// TIA Portal V20 export
FUNCTION_BLOCK "CallEquipment"   // FB43, LAD
TITLE = CallEquipment
// Template of an equipment module. This block contains the logic and futher calls (e.g. sequences, control modules, diagnostics etc.) of the equipment module.
// It can be used out of the box but also adapted to your own needs.
// stored: IsIECCheckEnabled true, MemoryReserve 100, Namespace Unit1.Em4, SetENOAutomatically true
   VAR_INPUT
      ZoneOperationEnable { ExternalWritable := 'False'} : "LWONIK_typeSafetyZoneManualOperation";
      unitEnableControlInterfaces { ExternalWritable := 'False'} : "LAF_typeEnableControlInterfaces";
      commandExcute { ExternalWritable := 'False'} : Bool;
   END_VAR
   VAR_IN_OUT
      unitStatus : "LAF_typeUnitStatus";   // Current unit status o be used in this EM
      emFeedback : "LUC_typeEmFeedback";   // Feedback of the EM to the Unit
      unitAlarmDB : "LAF_typeAlarms";   // Summarized EM Alarms for the Unit
   END_VAR
   VAR
      instSequence { ExternalWritable := 'False'} : "Unit1.Em4.Sequence_1_Cutter";
      instCutterInitializedJob1 { ExternalWritable := 'False'} : "LAF_SelectJob";
      instCutterCycleJob2 { S7_SetPoint := 'True'} : "LAF_SelectJob";
      instCmCompensatorAxisZ { ExternalWritable := 'False'} : "LBC_AxisControl_TecPlcCn";
      instCmFeedingRollAxisB { ExternalWritable := 'False'} : "LBC_AxisControl_TecPlcCn";
      instCmElectrodeCutterAxisZ { ExternalWritable := 'False'} : "LBC_AxisControl_TecPlcCn";
      instCmPositionMovingAxisX { ExternalWritable := 'False'} : "LBC_Axis64Pos_TecPlcCn";
      instCmFeederCylinderUpDown { ExternalWritable := 'False'} : "LBC_TwoWayActuatorCn";
      instCmCompensatorSafetyPinIdlePosition { ExternalWritable := 'False'} : "LBC_DigitalSignalCn";
      instCmTabDetectSensor { ExternalWritable := 'False'} : "LBC_DigitalSignalCn";
      instCmTapeDetectSensor { ExternalWritable := 'False'} : "LBC_DigitalSignalCn";
      instCutterEpcAnalogInput { ExternalWritable := 'False'} : "LBC_AnalogInputCn";
      instCompensatorAxisControlInterlockSummary { ExternalWritable := 'False'} : "LER_AxisControl_InterlockSummary";
      instFeedingRollAxisControlInterlockSummary { ExternalWritable := 'False'} : "LER_AxisControl_InterlockSummary";
      instCutterAxisControlInterlockSummary { ExternalWritable := 'False'} : "LER_AxisControl_InterlockSummary";
      instPostionMovingAxisControlInterlockSummary { ExternalWritable := 'False'} : "LER_Axis64Pos_InterlockSummary";
      instServoTorqueCal_DR3 { ExternalWritable := 'False'} : "LER_ServoTorqueCal";
      instServoTorqueCal_DR4 { ExternalWritable := 'False'} : "LER_ServoTorqueCal";
      instServoTorqueCal_DR5 { ExternalWritable := 'False'} : "LER_ServoTorqueCal";
      instServoTorqueCal_DR6 { ExternalWritable := 'False'} : "LER_ServoTorqueCal";
      instLDrv701ControlCompensatorAxisZ { ExternalWritable := 'False'} : "LDrvSafe_SinaTlg701Control";   // Drive Telegram Function Library
      instLDrv701StatusCompensatorAxisZ { ExternalWritable := 'False'} : "LDrvSafe_SinaTlg701Status";   // Drive Telegram Function Library
      instLDrv701ControlFeedingRollAxisB { ExternalWritable := 'False'} : "LDrvSafe_SinaTlg701Control";   // Drive Telegram Function Library
      instLDrv701StatusFeedingRollAxisB { ExternalWritable := 'False'} : "LDrvSafe_SinaTlg701Status";   // Drive Telegram Function Library
      instLDrv701ControlElectrodeCutterAxisZ { ExternalWritable := 'False'} : "LDrvSafe_SinaTlg701Control";   // Drive Telegram Function Library
      instLDrv701StatusElectrodeCutterAxisZ { ExternalWritable := 'False'} : "LDrvSafe_SinaTlg701Status";   // Drive Telegram Function Library
      instLDrv701ControlPositionMovingAxisX { ExternalWritable := 'False'} : "LDrvSafe_SinaTlg701Control";   // Drive Telegram Function Library
      instLDrv701StatusPositionMovingAxisX { ExternalWritable := 'False'} : "LDrvSafe_SinaTlg701Status";   // Drive Telegram Function Library
      statUnitStatus { ExternalWritable := 'False'} : "LAF_typeUnitStatus";   // Unit Status used in this EM
      statAllBrakeTest { ExternalWritable := 'False'} : "LER_typeBrakeTestUnitCommands";
      instManageAlarms { ExternalWritable := 'False'} : "LAF_ManageAlarms";
      instEventsPFE { S7_SetPoint := 'True'} : "Unit1.Em4.EventsPFE";
      statPulse { ExternalWritable := 'False'} : Array[0..99] of Bool;
      statTonTimer { ExternalWritable := 'False'} : Array[0..99] of TON_TIME;
      statTofTimer { ExternalWritable := 'False'} : Array[0..99] of TOF_TIME;
      statEnableManualCmds { ExternalWritable := 'False'} : Bool;
      EndOfCycle_Complete { ExternalWritable := 'False'} : Bool;
   END_VAR
   VAR_TEMP
      tempScInProduction : Bool;   // Mode Production and StateComplete
      tempScNoProduction : Bool;   // Mode Manual and StateComplete
   END_VAR
   VAR CONSTANT
      TO_DO_INSERT_PRECONDITIONS_HERE : Bool := TRUE;   // Template : Add em specific conditions here
      NO_JOB : DInt;   // No job
      TRUE : Bool := TRUE;
      FALSE : Bool := FALSE;
      "acc/dccTime" : LReal := 3.0;
      JerkTime : LReal := 0.0;
      INIT_POSITION_NUMBER : SInt := -1;
      MIN_POSITION_NUMBER : SInt;
   END_VAR
   VAR_TEMP   // added for the SCL form of the ladder/FBD networks
      _w1 : Bool;
      _w2 : Bool;
      _w3 : Bool;
      _w4 : Bool;
      _w5 : Bool;
      _w6 : Bool;
      _w7 : Bool;
      _w8 : Bool;
      _w9 : Bool;
      _w10 : Bool;
      _w11 : Bool;
      _w12 : Bool;
      _w13 : Bool;
      _w14 : Bool;
      _w15 : Bool;
      _w16 : Bool;
   END_VAR
BEGIN

REGION Network 1: BLOCK INFO HEADER
   // (company) / (C) Copyright (year)
   // ---------------------------------------------------------------------------------
   // Title:                             (Title of this block)
   // Comment/Function: (that is implemented in the block)
   // Library/Family:           (that the source is dedicated to)
   // Author:                        (department / person in charge / contact)
   // Target System:          (test system with FW version)
   // Engineering:              TIA Portal (SW version)
   // Restrictions:               (OB types, etc.)
   // Requirements:           (hardware, technological package, etc.)
   // ---------------------------------------------------------------------------------
   // Change log table:
   // Version          | Date             | Signature      | Expert in charge  | Changes applied ------------------------|----------------------|-------------------------|--------------------------------|-----------------------
   // 001.000.000 | yyyy-mm-dd | 0x00000000 | (name of expert) | First released version
END_REGION

REGION Network 2: DESCRIPTION
   // This is a template block provided by the Automation Framework. It can be used to create an own project.
   // The Block Info Header is prepared to put in your own data.
   // Description of the block could be added here and the docu created by Code2Docu.
END_REGION

REGION Network 3: ******************** Unit Input ********************
END_REGION

REGION Network 4: Em Nodes Brake Test
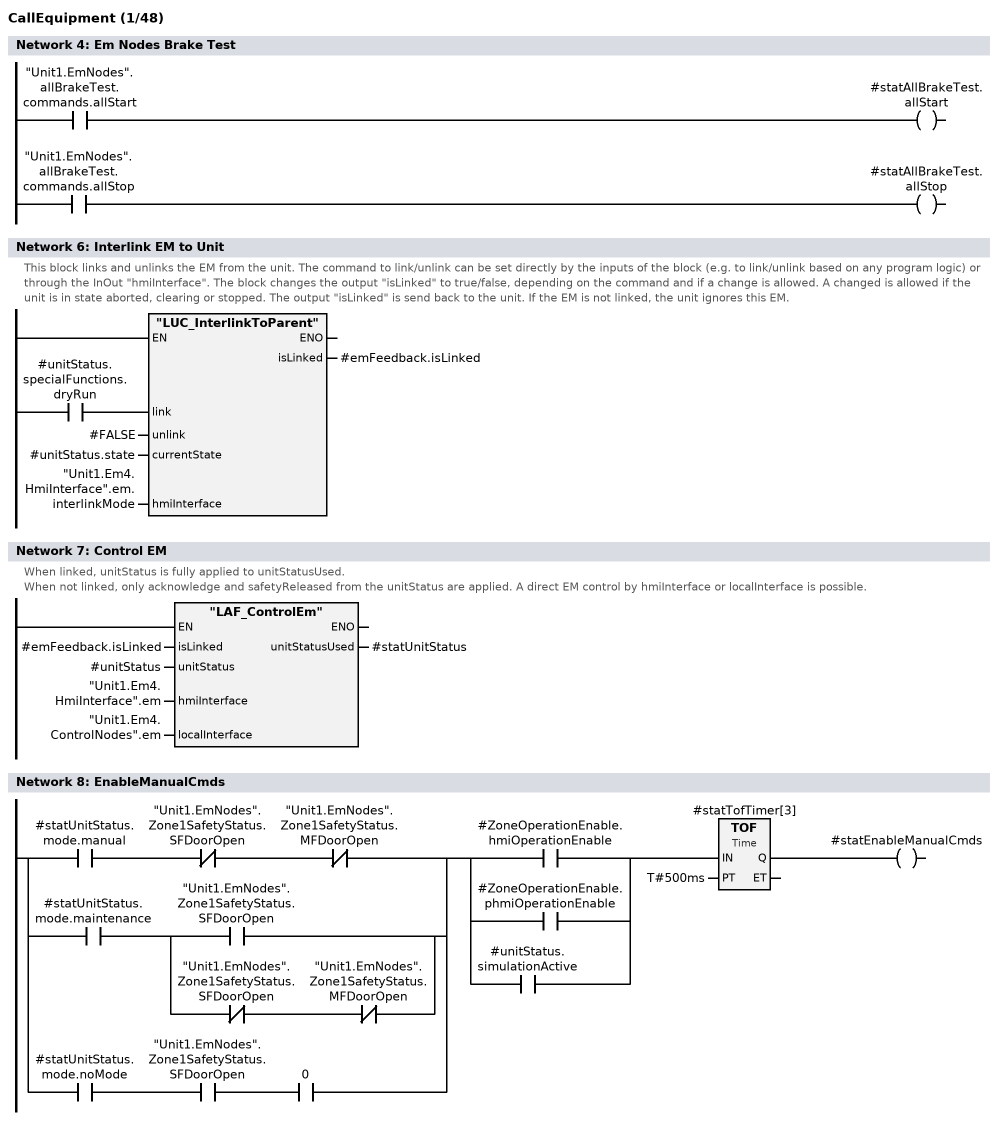
   RUNG wire#powerrail
      Contact( "Unit1.EmNodes".allBrakeTest.commands.allStart )
      Coil( #statAllBrakeTest.allStart )
   END_RUNG
   RUNG wire#powerrail
      Contact( "Unit1.EmNodes".allBrakeTest.commands.allStop )
      Coil( #statAllBrakeTest.allStop )
   END_RUNG
   // the same network as SCL:
   #statAllBrakeTest.allStart := "Unit1.EmNodes".allBrakeTest.commands.allStart;
   #statAllBrakeTest.allStop := "Unit1.EmNodes".allBrakeTest.commands.allStop;
END_REGION

REGION Network 5: ******************** Equipment Control ********************
END_REGION

REGION Network 6: Interlink EM to Unit
   // This block links and unlinks the EM from the unit. The command to link/unlink can be set directly by the inputs of the block (e.g. to link/unlink based on any program logic) or through the InOut "hmiInterface". The block changes the output "isLinked" to true/false, depending on the command and if a change is allowed. A changed is allowed if the unit is in state aborted, clearing or stopped. The output "isLinked" is send back to the unit. If the EM is not linked, the unit ignores this EM.
   RUNG wire#powerrail
      "LUC_InterlinkToParent"(link := wire#w1, unlink := #FALSE, currentState := #unitStatus.state, hmiInterface := "Unit1.Em4.HmiInterface".em.interlinkMode, isLinked => #emFeedback.isLinked)
   END_RUNG
   RUNG wire#powerrail
      Contact( #unitStatus.specialFunctions.dryRun )
   END_RUNG wire#w1
   // the same network as SCL:
   "LUC_InterlinkToParent"(link := #unitStatus.specialFunctions.dryRun,
                           unlink := #FALSE,
                           currentState := #unitStatus.state,
                           hmiInterface := "Unit1.Em4.HmiInterface".em.interlinkMode,
                           isLinked => #emFeedback.isLinked);
END_REGION

REGION Network 7: Control EM
   // When linked, unitStatus is fully applied to unitStatusUsed.
   // When not linked, only acknowledge and safetyReleased from the unitStatus are applied. A direct EM control by hmiInterface or localInterface is possible.
   RUNG wire#powerrail
      "LAF_ControlEm"(isLinked := #emFeedback.isLinked, unitStatus := #unitStatus, hmiInterface := "Unit1.Em4.HmiInterface".em, localInterface := "Unit1.Em4.ControlNodes".em, unitStatusUsed => #statUnitStatus)
   END_RUNG
   // the same network as SCL:
   "LAF_ControlEm"(isLinked := #emFeedback.isLinked,
                   unitStatus := #unitStatus,
                   hmiInterface := "Unit1.Em4.HmiInterface".em,
                   localInterface := "Unit1.Em4.ControlNodes".em,
                   unitStatusUsed => #statUnitStatus);
END_REGION

REGION Network 8: EnableManualCmds
   RUNG wire#powerrail
      Contact( #statUnitStatus.mode.manual )
      I_Contact( "Unit1.EmNodes".Zone1SafetyStatus.SFDoorOpen )
      I_Contact( "Unit1.EmNodes".Zone1SafetyStatus.MFDoorOpen )
      wire#w1
      Contact( #ZoneOperationEnable.hmiOperationEnable )
      wire#w3
      { S7_Templates := "time_type := Time" } #statTofTimer[3].TOF(pt := T#500ms, et =>)
      Coil( #statEnableManualCmds )
   END_RUNG
   RUNG wire#powerrail
      Contact( #statUnitStatus.mode.maintenance )
      wire#w2
      Contact( "Unit1.EmNodes".Zone1SafetyStatus.SFDoorOpen )
   END_RUNG wire#w1
   RUNG wire#w2
      I_Contact( "Unit1.EmNodes".Zone1SafetyStatus.SFDoorOpen )
      I_Contact( "Unit1.EmNodes".Zone1SafetyStatus.MFDoorOpen )
   END_RUNG wire#w1
   RUNG wire#powerrail
      Contact( #statUnitStatus.mode.noMode )
      Contact( "Unit1.EmNodes".Zone1SafetyStatus.SFDoorOpen )
      Contact( 0 )
   END_RUNG wire#w1
   RUNG wire#w1
      Contact( #ZoneOperationEnable.phmiOperationEnable )
   END_RUNG wire#w3
   RUNG wire#w1
      Contact( #unitStatus.simulationActive )
   END_RUNG wire#w3
   // the same network as SCL:
   #statTofTimer[3].TOF(IN := ((#statUnitStatus.mode.manual AND NOT "Unit1.EmNodes".Zone1SafetyStatus.SFDoorOpen AND NOT "Unit1.EmNodes".Zone1SafetyStatus.MFDoorOpen) OR (#statUnitStatus.mode.maintenance AND ("Unit1.EmNodes".Zone1SafetyStatus.SFDoorOpen OR (NOT "Unit1.EmNodes".Zone1SafetyStatus.SFDoorOpen AND NOT "Unit1.EmNodes".Zone1SafetyStatus.MFDoorOpen))) OR (#statUnitStatus.mode.noMode AND "Unit1.EmNodes".Zone1SafetyStatus.SFDoorOpen AND 0)) AND (#ZoneOperationEnable.hmiOperationEnable OR #ZoneOperationEnable.phmiOperationEnable OR #unitStatus.simulationActive),
                        PT := T#500ms);
   #statEnableManualCmds := #statTofTimer[3].Q;
END_REGION

REGION Network 9: Alarms Disabled
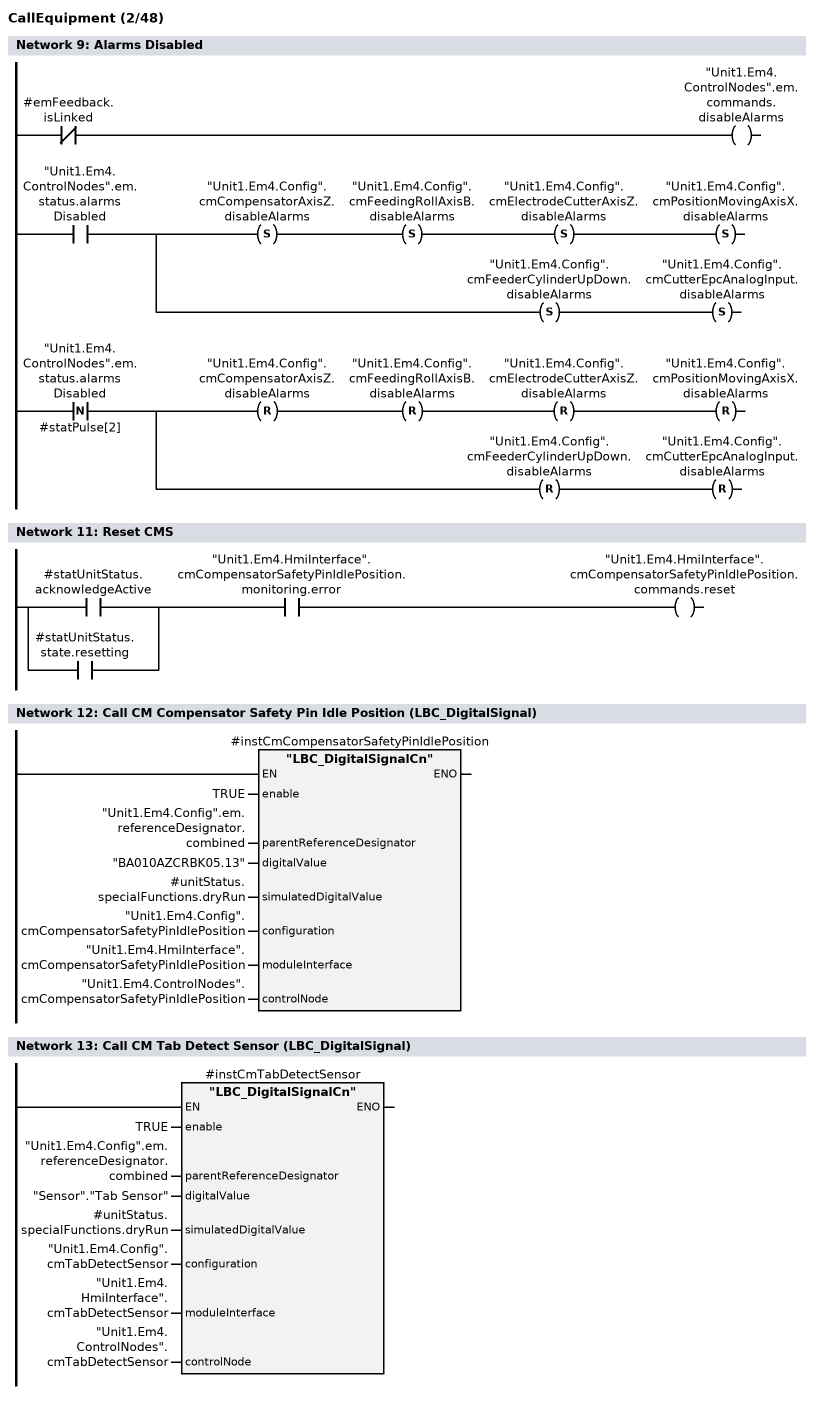
   RUNG wire#powerrail
      I_Contact( #emFeedback.isLinked )
      Coil( "Unit1.Em4.ControlNodes".em.commands.disableAlarms )
   END_RUNG
   RUNG wire#powerrail
      Contact( "Unit1.Em4.ControlNodes".em.status.alarmsDisabled )
      wire#w1
      S_Coil( "Unit1.Em4.Config".cmCompensatorAxisZ.disableAlarms )
      S_Coil( "Unit1.Em4.Config".cmFeedingRollAxisB.disableAlarms )
      S_Coil( "Unit1.Em4.Config".cmElectrodeCutterAxisZ.disableAlarms )
      S_Coil( "Unit1.Em4.Config".cmPositionMovingAxisX.disableAlarms )
   END_RUNG
   RUNG wire#w1
      S_Coil( "Unit1.Em4.Config".cmFeederCylinderUpDown.disableAlarms )
      S_Coil( "Unit1.Em4.Config".cmCutterEpcAnalogInput.disableAlarms )
   END_RUNG
   RUNG wire#powerrail
      N_Contact(operand := "Unit1.Em4.ControlNodes".em.status.alarmsDisabled, bit := #statPulse[2])
      wire#w2
      R_Coil( "Unit1.Em4.Config".cmCompensatorAxisZ.disableAlarms )
      R_Coil( "Unit1.Em4.Config".cmFeedingRollAxisB.disableAlarms )
      R_Coil( "Unit1.Em4.Config".cmElectrodeCutterAxisZ.disableAlarms )
      R_Coil( "Unit1.Em4.Config".cmPositionMovingAxisX.disableAlarms )
   END_RUNG
   RUNG wire#w2
      R_Coil( "Unit1.Em4.Config".cmFeederCylinderUpDown.disableAlarms )
      R_Coil( "Unit1.Em4.Config".cmCutterEpcAnalogInput.disableAlarms )
   END_RUNG
   // the same network as SCL:
   "Unit1.Em4.ControlNodes".em.commands.disableAlarms := NOT #emFeedback.isLinked;
   IF "Unit1.Em4.ControlNodes".em.status.alarmsDisabled THEN
       "Unit1.Em4.Config".cmCompensatorAxisZ.disableAlarms := TRUE;
       "Unit1.Em4.Config".cmFeedingRollAxisB.disableAlarms := TRUE;
       "Unit1.Em4.Config".cmElectrodeCutterAxisZ.disableAlarms := TRUE;
       "Unit1.Em4.Config".cmPositionMovingAxisX.disableAlarms := TRUE;
       "Unit1.Em4.Config".cmFeederCylinderUpDown.disableAlarms := TRUE;
       "Unit1.Em4.Config".cmCutterEpcAnalogInput.disableAlarms := TRUE;
   END_IF;
   #_w1 := NOT "Unit1.Em4.ControlNodes".em.status.alarmsDisabled AND #statPulse[2];   // falling edge of "Unit1.Em4.ControlNodes".em.status.alarmsDisabled
   #statPulse[2] := "Unit1.Em4.ControlNodes".em.status.alarmsDisabled;
   IF #_w1 THEN
       "Unit1.Em4.Config".cmCompensatorAxisZ.disableAlarms := FALSE;
       "Unit1.Em4.Config".cmFeedingRollAxisB.disableAlarms := FALSE;
       "Unit1.Em4.Config".cmElectrodeCutterAxisZ.disableAlarms := FALSE;
       "Unit1.Em4.Config".cmPositionMovingAxisX.disableAlarms := FALSE;
       "Unit1.Em4.Config".cmFeederCylinderUpDown.disableAlarms := FALSE;
       "Unit1.Em4.Config".cmCutterEpcAnalogInput.disableAlarms := FALSE;
   END_IF;
END_REGION

REGION Network 10: ******************** Control Modules (Sensors) ********************
   // Call control modules that are sensors before the em logic (jobs and sequence), so that the latest value is used in the logic.
END_REGION

REGION Network 11: Reset CMS
   RUNG wire#powerrail
      Contact( #statUnitStatus.acknowledgeActive )
      wire#w1
      Contact( "Unit1.Em4.HmiInterface".cmCompensatorSafetyPinIdlePosition.monitoring.error )
      Coil( "Unit1.Em4.HmiInterface".cmCompensatorSafetyPinIdlePosition.commands.reset )
   END_RUNG
   RUNG wire#powerrail
      Contact( #statUnitStatus.state.resetting )
   END_RUNG wire#w1
   // the same network as SCL:
   "Unit1.Em4.HmiInterface".cmCompensatorSafetyPinIdlePosition.commands.reset := (#statUnitStatus.acknowledgeActive OR #statUnitStatus.state.resetting) AND "Unit1.Em4.HmiInterface".cmCompensatorSafetyPinIdlePosition.monitoring.error;
END_REGION

REGION Network 12: Call CM Compensator Safety Pin Idle Position (LBC_DigitalSignal)
   RUNG wire#powerrail
      #instCmCompensatorSafetyPinIdlePosition(enable := TRUE, parentReferenceDesignator := "Unit1.Em4.Config".em.referenceDesignator.combined, digitalValue := "BA010AZCRBK05.13", simulatedDigitalValue := #unitStatus.specialFunctions.dryRun, configuration := "Unit1.Em4.Config".cmCompensatorSafetyPinIdlePosition, moduleInterface := "Unit1.Em4.HmiInterface".cmCompensatorSafetyPinIdlePosition, controlNode := "Unit1.Em4.ControlNodes".cmCompensatorSafetyPinIdlePosition)
   END_RUNG
   // the same network as SCL:
   #instCmCompensatorSafetyPinIdlePosition(enable := TRUE,   // "LBC_DigitalSignalCn"
                           parentReferenceDesignator := "Unit1.Em4.Config".em.referenceDesignator.combined,
                           digitalValue := "BA010AZCRBK05.13",
                           simulatedDigitalValue := #unitStatus.specialFunctions.dryRun,
                           configuration := "Unit1.Em4.Config".cmCompensatorSafetyPinIdlePosition,
                           moduleInterface := "Unit1.Em4.HmiInterface".cmCompensatorSafetyPinIdlePosition,
                           controlNode := "Unit1.Em4.ControlNodes".cmCompensatorSafetyPinIdlePosition);
END_REGION

REGION Network 13: Call CM Tab Detect Sensor (LBC_DigitalSignal)
   RUNG wire#powerrail
      #instCmTabDetectSensor(enable := TRUE, parentReferenceDesignator := "Unit1.Em4.Config".em.referenceDesignator.combined, digitalValue := "Sensor"."Tab Sensor", simulatedDigitalValue := #unitStatus.specialFunctions.dryRun, configuration := "Unit1.Em4.Config".cmTabDetectSensor, moduleInterface := "Unit1.Em4.HmiInterface".cmTabDetectSensor, controlNode := "Unit1.Em4.ControlNodes".cmTabDetectSensor)
   END_RUNG
   // the same network as SCL:
   #instCmTabDetectSensor(enable := TRUE,   // "LBC_DigitalSignalCn"
                          parentReferenceDesignator := "Unit1.Em4.Config".em.referenceDesignator.combined,
                          digitalValue := "Sensor"."Tab Sensor",
                          simulatedDigitalValue := #unitStatus.specialFunctions.dryRun,
                          configuration := "Unit1.Em4.Config".cmTabDetectSensor,
                          moduleInterface := "Unit1.Em4.HmiInterface".cmTabDetectSensor,
                          controlNode := "Unit1.Em4.ControlNodes".cmTabDetectSensor);
END_REGION

REGION Network 14: Call CM Tape Detect Sensor (LBC_DigitalSignal)
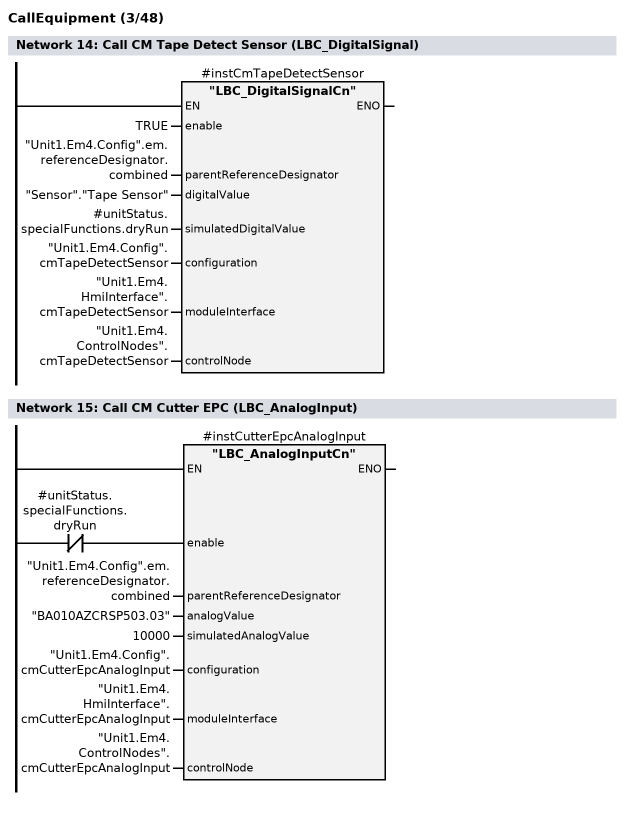
   RUNG wire#powerrail
      #instCmTapeDetectSensor(enable := TRUE, parentReferenceDesignator := "Unit1.Em4.Config".em.referenceDesignator.combined, digitalValue := "Sensor"."Tape Sensor", simulatedDigitalValue := #unitStatus.specialFunctions.dryRun, configuration := "Unit1.Em4.Config".cmTapeDetectSensor, moduleInterface := "Unit1.Em4.HmiInterface".cmTapeDetectSensor, controlNode := "Unit1.Em4.ControlNodes".cmTapeDetectSensor)
   END_RUNG
   // the same network as SCL:
   #instCmTapeDetectSensor(enable := TRUE,   // "LBC_DigitalSignalCn"
                           parentReferenceDesignator := "Unit1.Em4.Config".em.referenceDesignator.combined,
                           digitalValue := "Sensor"."Tape Sensor",
                           simulatedDigitalValue := #unitStatus.specialFunctions.dryRun,
                           configuration := "Unit1.Em4.Config".cmTapeDetectSensor,
                           moduleInterface := "Unit1.Em4.HmiInterface".cmTapeDetectSensor,
                           controlNode := "Unit1.Em4.ControlNodes".cmTapeDetectSensor);
END_REGION

REGION Network 15: Call CM Cutter EPC (LBC_AnalogInput)
   RUNG wire#powerrail
      #instCutterEpcAnalogInput(enable := wire#w1, parentReferenceDesignator := "Unit1.Em4.Config".em.referenceDesignator.combined, analogValue := "BA010AZCRSP503.03", simulatedAnalogValue := 10000, configuration := "Unit1.Em4.Config".cmCutterEpcAnalogInput, moduleInterface := "Unit1.Em4.HmiInterface".cmCutterEpcAnalogInput, controlNode := "Unit1.Em4.ControlNodes".cmCutterEpcAnalogInput)
   END_RUNG
   RUNG wire#powerrail
      I_Contact( #unitStatus.specialFunctions.dryRun )
   END_RUNG wire#w1
   // the same network as SCL:
   #instCutterEpcAnalogInput(enable := NOT #unitStatus.specialFunctions.dryRun,   // "LBC_AnalogInputCn"
                           parentReferenceDesignator := "Unit1.Em4.Config".em.referenceDesignator.combined,
                           analogValue := "BA010AZCRSP503.03",
                           simulatedAnalogValue := 10000,
                           configuration := "Unit1.Em4.Config".cmCutterEpcAnalogInput,
                           moduleInterface := "Unit1.Em4.HmiInterface".cmCutterEpcAnalogInput,
                           controlNode := "Unit1.Em4.ControlNodes".cmCutterEpcAnalogInput);
END_REGION

REGION Network 16: ******************** Equipment Logic ********************
END_REGION

REGION Network 17: Map Unit Status to Sequence Status [1] Cutter
   // This block maps the unit status to the seuqnce status. Thus, it controls the sequence depending on the unit status. E.g. it sets the sequence to automatic when the unit state is in productions. This blocks work perfectly with the sequences provided in the AF. 
   // This typed block (MapUnitStatusToSequence) could be adjusted to specific application requirements or if other, user-defined sequences are used.
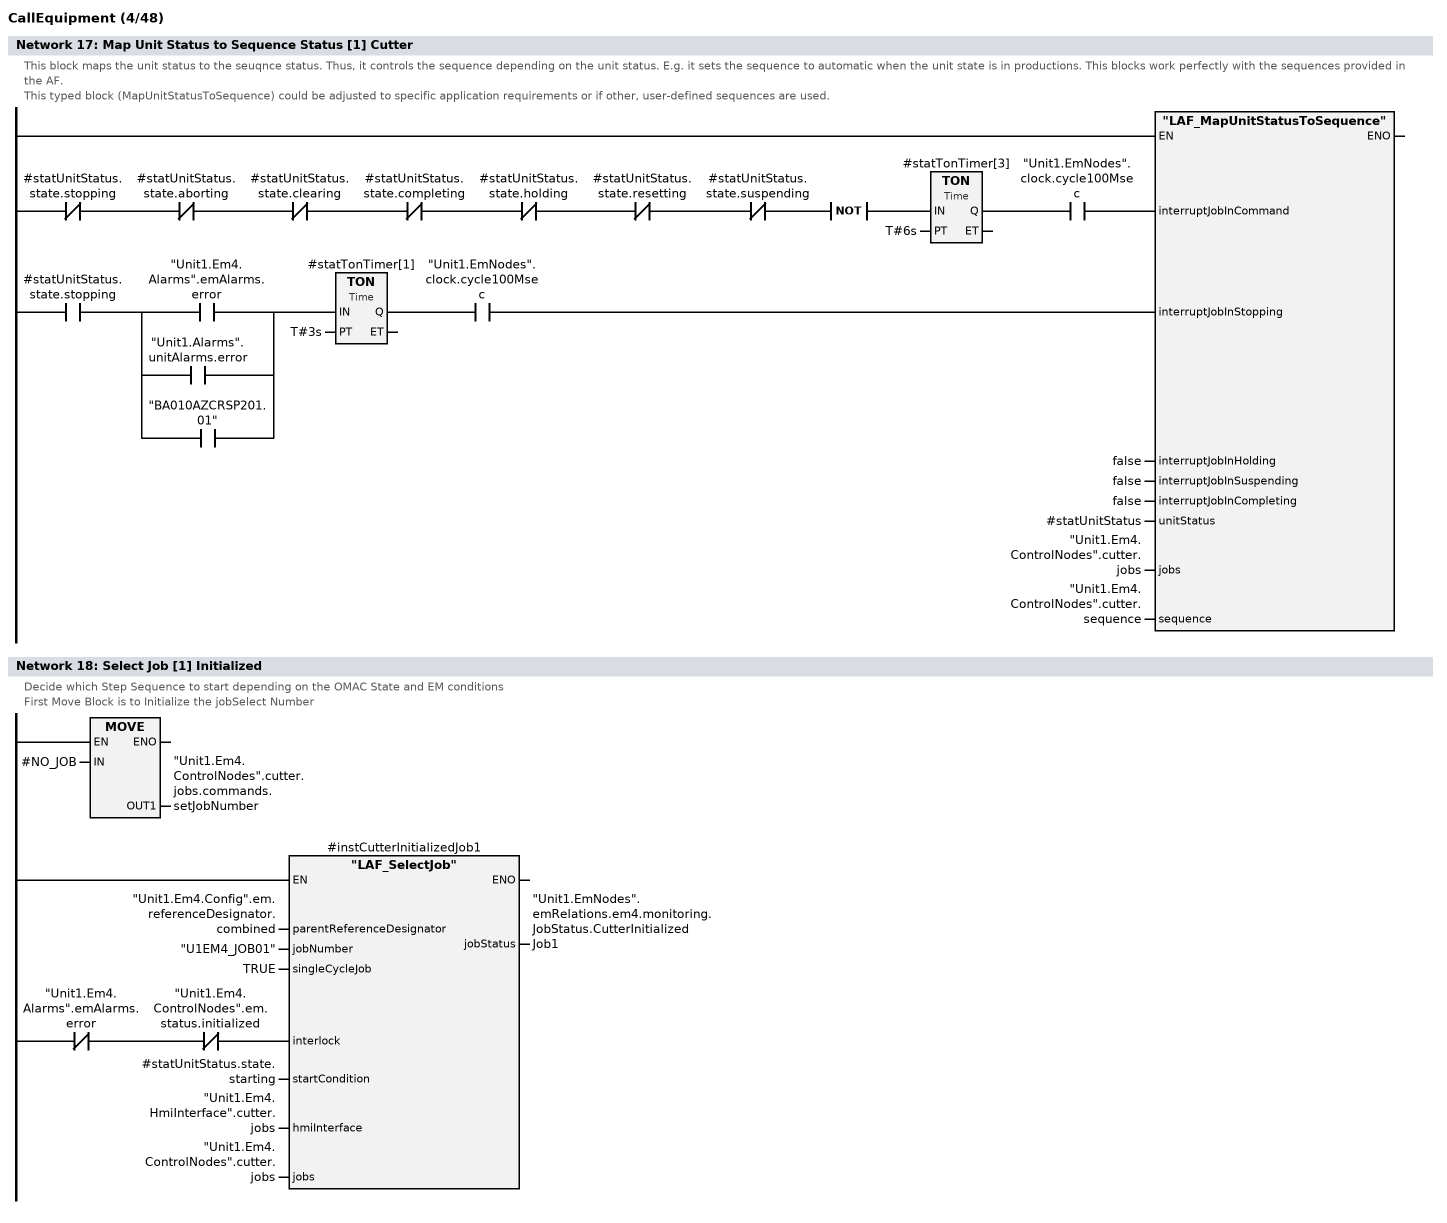
   RUNG wire#powerrail
      "LAF_MapUnitStatusToSequence"(interruptJobInCommand := wire#w1, interruptJobInStopping := wire#w4, interruptJobInHolding := false, interruptJobInSuspending := false, interruptJobInCompleting := false, unitStatus := #statUnitStatus, jobs := "Unit1.Em4.ControlNodes".cutter.jobs, sequence := "Unit1.Em4.ControlNodes".cutter.sequence)
   END_RUNG
   RUNG wire#powerrail
      I_Contact( #statUnitStatus.state.stopping )
      I_Contact( #statUnitStatus.state.aborting )
      I_Contact( #statUnitStatus.state.clearing )
      I_Contact( #statUnitStatus.state.completing )
      I_Contact( #statUnitStatus.state.holding )
      I_Contact( #statUnitStatus.state.resetting )
      I_Contact( #statUnitStatus.state.suspending )
      Not()
      { S7_Templates := "time_type := Time" } #statTonTimer[3].TON(pt := T#6s, et =>)
      Contact( "Unit1.EmNodes".clock.cycle100Msec )
   END_RUNG wire#w1
   RUNG wire#powerrail
      Contact( #statUnitStatus.state.stopping )
      wire#w2
      Contact( "Unit1.Em4.Alarms".emAlarms.error )
      wire#w3
      { S7_Templates := "time_type := Time" } #statTonTimer[1].TON(pt := T#3s, et =>)
      Contact( "Unit1.EmNodes".clock.cycle100Msec )
   END_RUNG wire#w4
   RUNG wire#w2
      Contact( "Unit1.Alarms".unitAlarms.error )
   END_RUNG wire#w3
   RUNG wire#w2
      Contact( "BA010AZCRSP201.01" )
   END_RUNG wire#w3
   // the same network as SCL:
   #statTonTimer[3].TON(IN := NOT (NOT #statUnitStatus.state.stopping AND NOT #statUnitStatus.state.aborting AND NOT #statUnitStatus.state.clearing AND NOT #statUnitStatus.state.completing AND NOT #statUnitStatus.state.holding AND NOT #statUnitStatus.state.resetting AND NOT #statUnitStatus.state.suspending),
                        PT := T#6s);
   #_w1 := #statTonTimer[3].Q AND "Unit1.EmNodes".clock.cycle100Msec;
   #statTonTimer[1].TON(IN := #statUnitStatus.state.stopping AND ("Unit1.Em4.Alarms".emAlarms.error OR "Unit1.Alarms".unitAlarms.error OR "BA010AZCRSP201.01"),
                        PT := T#3s);
   "LAF_MapUnitStatusToSequence"(interruptJobInCommand := #_w1,
                           interruptJobInStopping := #statTonTimer[1].Q AND "Unit1.EmNodes".clock.cycle100Msec,
                           interruptJobInHolding := false,
                           interruptJobInSuspending := false,
                           interruptJobInCompleting := false,
                           unitStatus := #statUnitStatus,
                           jobs := "Unit1.Em4.ControlNodes".cutter.jobs,
                           sequence := "Unit1.Em4.ControlNodes".cutter.sequence);
END_REGION

REGION Network 18: Select Job [1] Initialized
   // Decide which Step Sequence to start depending on the OMAC State and EM conditions
   // First Move Block is to Initialize the jobSelect Number
   RUNG wire#powerrail
      Move(in := #NO_JOB, out1 => "Unit1.Em4.ControlNodes".cutter.jobs.commands.setJobNumber)
   END_RUNG
   RUNG wire#powerrail
      #instCutterInitializedJob1(interlock := wire#w1, parentReferenceDesignator := "Unit1.Em4.Config".em.referenceDesignator.combined, jobNumber := "U1EM4_JOB01", singleCycleJob := TRUE, startCondition := #statUnitStatus.state.starting, hmiInterface := "Unit1.Em4.HmiInterface".cutter.jobs, jobs := "Unit1.Em4.ControlNodes".cutter.jobs, jobStatus => "Unit1.EmNodes".emRelations.em4.monitoring.JobStatus.CutterInitializedJob1)
   END_RUNG
   RUNG wire#powerrail
      I_Contact( "Unit1.Em4.Alarms".emAlarms.error )
      I_Contact( "Unit1.Em4.ControlNodes".em.status.initialized )
   END_RUNG wire#w1
   // the same network as SCL:
   "Unit1.Em4.ControlNodes".cutter.jobs.commands.setJobNumber := #NO_JOB;
   #instCutterInitializedJob1(parentReferenceDesignator := "Unit1.Em4.Config".em.referenceDesignator.combined,   // "LAF_SelectJob"
                           jobNumber := "U1EM4_JOB01",
                           singleCycleJob := TRUE,
                           interlock := NOT "Unit1.Em4.Alarms".emAlarms.error AND NOT "Unit1.Em4.ControlNodes".em.status.initialized,
                           startCondition := #statUnitStatus.state.starting,
                           hmiInterface := "Unit1.Em4.HmiInterface".cutter.jobs,
                           jobs := "Unit1.Em4.ControlNodes".cutter.jobs,
                           jobStatus => "Unit1.EmNodes".emRelations.em4.monitoring.JobStatus.CutterInitializedJob1);
END_REGION

REGION Network 19: Select Job [2] Cutter One Cycle(For Recovery)
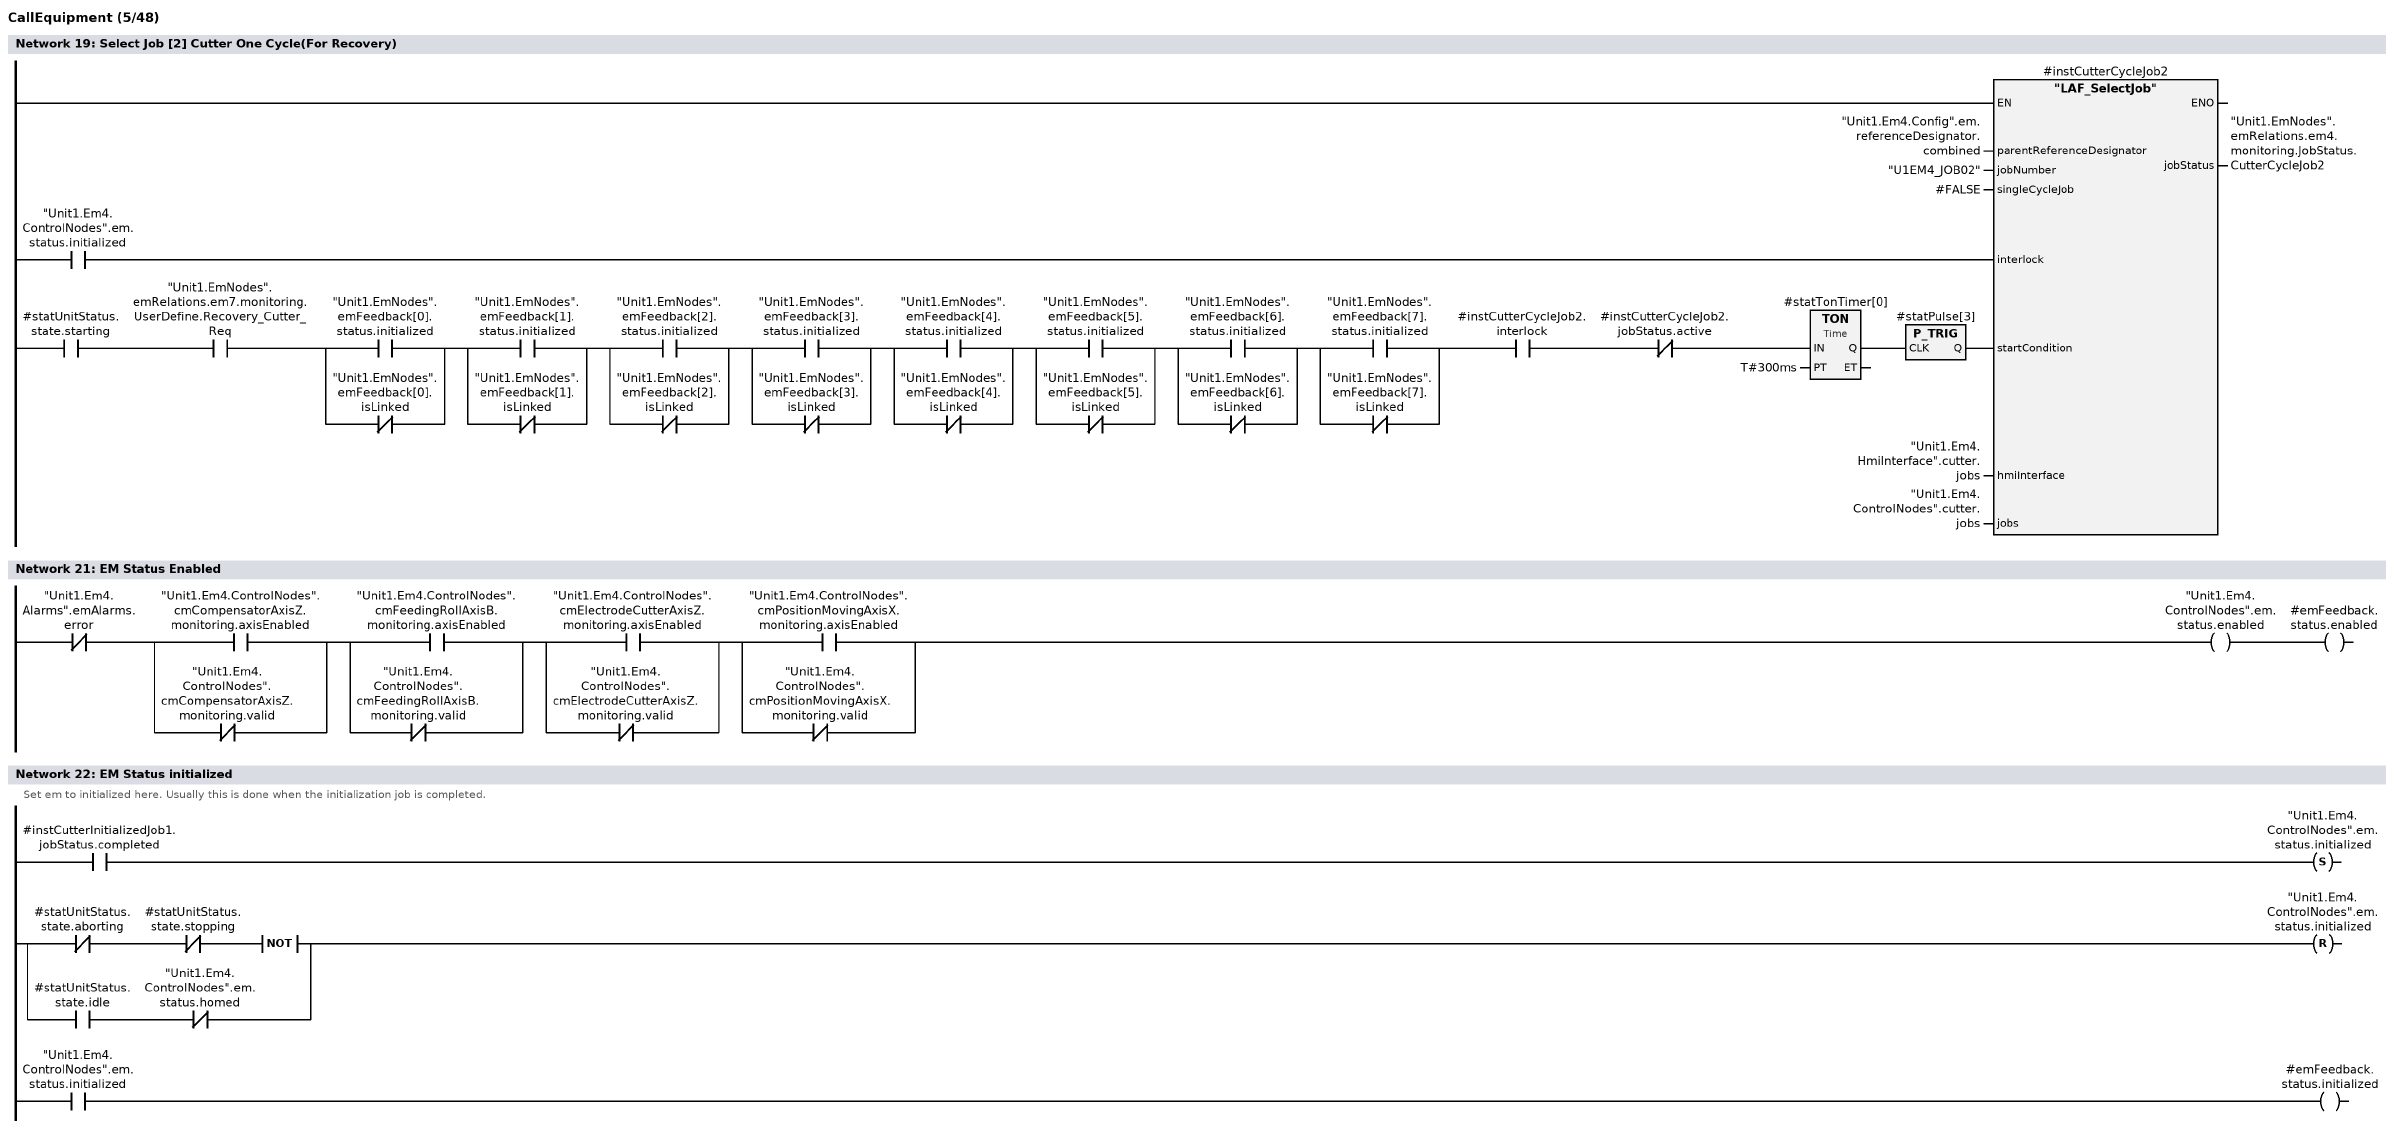
   RUNG wire#powerrail
      #instCutterCycleJob2(interlock := wire#w1, startCondition := wire#w11, parentReferenceDesignator := "Unit1.Em4.Config".em.referenceDesignator.combined, jobNumber := "U1EM4_JOB02", singleCycleJob := #FALSE, hmiInterface := "Unit1.Em4.HmiInterface".cutter.jobs, jobs := "Unit1.Em4.ControlNodes".cutter.jobs, jobStatus => "Unit1.EmNodes".emRelations.em4.monitoring.JobStatus.CutterCycleJob2)
   END_RUNG
   RUNG wire#powerrail
      Contact( "Unit1.Em4.ControlNodes".em.status.initialized )
   END_RUNG wire#w1
   RUNG wire#powerrail
      Contact( #statUnitStatus.state.starting )
      Contact( "Unit1.EmNodes".emRelations.em7.monitoring.UserDefine.Recovery_Cutter_Req )
      wire#w2
      Contact( "Unit1.EmNodes".emFeedback[0].status.initialized )
      wire#w3
      Contact( "Unit1.EmNodes".emFeedback[1].status.initialized )
      wire#w4
      Contact( "Unit1.EmNodes".emFeedback[2].status.initialized )
      wire#w5
      Contact( "Unit1.EmNodes".emFeedback[3].status.initialized )
      wire#w6
      Contact( "Unit1.EmNodes".emFeedback[4].status.initialized )
      wire#w7
      Contact( "Unit1.EmNodes".emFeedback[5].status.initialized )
      wire#w8
      Contact( "Unit1.EmNodes".emFeedback[6].status.initialized )
      wire#w9
      Contact( "Unit1.EmNodes".emFeedback[7].status.initialized )
      wire#w10
      Contact( #instCutterCycleJob2.interlock )
      I_Contact( #instCutterCycleJob2.jobStatus.active )
      { S7_Templates := "time_type := Time" } #statTonTimer[0].TON(pt := T#300ms, et =>)
      P_Trig( #statPulse[3] )
   END_RUNG wire#w11
   RUNG wire#w2
      I_Contact( "Unit1.EmNodes".emFeedback[0].isLinked )
   END_RUNG wire#w3
   RUNG wire#w3
      I_Contact( "Unit1.EmNodes".emFeedback[1].isLinked )
   END_RUNG wire#w4
   RUNG wire#w4
      I_Contact( "Unit1.EmNodes".emFeedback[2].isLinked )
   END_RUNG wire#w5
   RUNG wire#w5
      I_Contact( "Unit1.EmNodes".emFeedback[3].isLinked )
   END_RUNG wire#w6
   RUNG wire#w6
      I_Contact( "Unit1.EmNodes".emFeedback[4].isLinked )
   END_RUNG wire#w7
   RUNG wire#w7
      I_Contact( "Unit1.EmNodes".emFeedback[5].isLinked )
   END_RUNG wire#w8
   RUNG wire#w8
      I_Contact( "Unit1.EmNodes".emFeedback[6].isLinked )
   END_RUNG wire#w9
   RUNG wire#w9
      I_Contact( "Unit1.EmNodes".emFeedback[7].isLinked )
   END_RUNG wire#w10
   // the same network as SCL:
   #statTonTimer[0].TON(IN := #statUnitStatus.state.starting AND "Unit1.EmNodes".emRelations.em7.monitoring.UserDefine.Recovery_Cutter_Req AND ("Unit1.EmNodes".emFeedback[0].status.initialized OR NOT "Unit1.EmNodes".emFeedback[0].isLinked) AND ("Unit1.EmNodes".emFeedback[1].status.initialized OR NOT "Unit1.EmNodes".emFeedback[1].isLinked) AND ("Unit1.EmNodes".emFeedback[2].status.initialized OR NOT "Unit1.EmNodes".emFeedback[2].isLinked) AND ("Unit1.EmNodes".emFeedback[3].status.initialized OR NOT "Unit1.EmNodes".emFeedback[3].isLinked) AND ("Unit1.EmNodes".emFeedback[4].status.initialized OR NOT "Unit1.EmNodes".emFeedback[4].isLinked) AND ("Unit1.EmNodes".emFeedback[5].status.initialized OR NOT "Unit1.EmNodes".emFeedback[5].isLinked) AND ("Unit1.EmNodes".emFeedback[6].status.initialized OR NOT "Unit1.EmNodes".emFeedback[6].isLinked) AND ("Unit1.EmNodes".emFeedback[7].status.initialized OR NOT "Unit1.EmNodes".emFeedback[7].isLinked) AND #instCutterCycleJob2.interlock AND NOT #instCutterCycleJob2.jobStatus.active,
                        PT := T#300ms);
   #_w1 := #statTonTimer[0].Q AND NOT #statPulse[3];   // rising edge
   #statPulse[3] := #statTonTimer[0].Q;
   #instCutterCycleJob2(parentReferenceDesignator := "Unit1.Em4.Config".em.referenceDesignator.combined,   // "LAF_SelectJob"
                        jobNumber := "U1EM4_JOB02",
                        singleCycleJob := #FALSE,
                        interlock := "Unit1.Em4.ControlNodes".em.status.initialized,
                        startCondition := #_w1,
                        hmiInterface := "Unit1.Em4.HmiInterface".cutter.jobs,
                        jobs := "Unit1.Em4.ControlNodes".cutter.jobs,
                        jobStatus => "Unit1.EmNodes".emRelations.em4.monitoring.JobStatus.CutterCycleJob2);
END_REGION

REGION Network 20: Select Job Working Done
END_REGION

REGION Network 21: EM Status Enabled
   RUNG wire#powerrail
      I_Contact( "Unit1.Em4.Alarms".emAlarms.error )
      wire#w1
      Contact( "Unit1.Em4.ControlNodes".cmCompensatorAxisZ.monitoring.axisEnabled )
      wire#w2
      Contact( "Unit1.Em4.ControlNodes".cmFeedingRollAxisB.monitoring.axisEnabled )
      wire#w3
      Contact( "Unit1.Em4.ControlNodes".cmElectrodeCutterAxisZ.monitoring.axisEnabled )
      wire#w4
      Contact( "Unit1.Em4.ControlNodes".cmPositionMovingAxisX.monitoring.axisEnabled )
      wire#w5
      Coil( "Unit1.Em4.ControlNodes".em.status.enabled )
      Coil( #emFeedback.status.enabled )
   END_RUNG
   RUNG wire#w1
      I_Contact( "Unit1.Em4.ControlNodes".cmCompensatorAxisZ.monitoring.valid )
   END_RUNG wire#w2
   RUNG wire#w2
      I_Contact( "Unit1.Em4.ControlNodes".cmFeedingRollAxisB.monitoring.valid )
   END_RUNG wire#w3
   RUNG wire#w3
      I_Contact( "Unit1.Em4.ControlNodes".cmElectrodeCutterAxisZ.monitoring.valid )
   END_RUNG wire#w4
   RUNG wire#w4
      I_Contact( "Unit1.Em4.ControlNodes".cmPositionMovingAxisX.monitoring.valid )
   END_RUNG wire#w5
   // the same network as SCL:
   "Unit1.Em4.ControlNodes".em.status.enabled := NOT "Unit1.Em4.Alarms".emAlarms.error AND ("Unit1.Em4.ControlNodes".cmCompensatorAxisZ.monitoring.axisEnabled OR NOT "Unit1.Em4.ControlNodes".cmCompensatorAxisZ.monitoring.valid) AND ("Unit1.Em4.ControlNodes".cmFeedingRollAxisB.monitoring.axisEnabled OR NOT "Unit1.Em4.ControlNodes".cmFeedingRollAxisB.monitoring.valid) AND ("Unit1.Em4.ControlNodes".cmElectrodeCutterAxisZ.monitoring.axisEnabled OR NOT "Unit1.Em4.ControlNodes".cmElectrodeCutterAxisZ.monitoring.valid) AND ("Unit1.Em4.ControlNodes".cmPositionMovingAxisX.monitoring.axisEnabled OR NOT "Unit1.Em4.ControlNodes".cmPositionMovingAxisX.monitoring.valid);
   #emFeedback.status.enabled := "Unit1.Em4.ControlNodes".em.status.enabled;
END_REGION

REGION Network 22: EM Status initialized
   // Set em to initialized here. Usually this is done when the initialization job is completed.
   RUNG wire#powerrail
      Contact( #instCutterInitializedJob1.jobStatus.completed )
      S_Coil( "Unit1.Em4.ControlNodes".em.status.initialized )
   END_RUNG
   RUNG wire#powerrail
      I_Contact( #statUnitStatus.state.aborting )
      I_Contact( #statUnitStatus.state.stopping )
      Not()
      wire#w1
      R_Coil( "Unit1.Em4.ControlNodes".em.status.initialized )
   END_RUNG
   RUNG wire#powerrail
      Contact( #statUnitStatus.state.idle )
      I_Contact( "Unit1.Em4.ControlNodes".em.status.homed )
   END_RUNG wire#w1
   RUNG wire#powerrail
      Contact( "Unit1.Em4.ControlNodes".em.status.initialized )
      Coil( #emFeedback.status.initialized )
   END_RUNG
   // the same network as SCL:
   IF #instCutterInitializedJob1.jobStatus.completed THEN
       "Unit1.Em4.ControlNodes".em.status.initialized := TRUE;
   END_IF;
   IF NOT (NOT #statUnitStatus.state.aborting AND NOT #statUnitStatus.state.stopping) OR (#statUnitStatus.state.idle AND NOT "Unit1.Em4.ControlNodes".em.status.homed) THEN
       "Unit1.Em4.ControlNodes".em.status.initialized := FALSE;
   END_IF;
   #emFeedback.status.initialized := "Unit1.Em4.ControlNodes".em.status.initialized;
END_REGION

REGION Network 23: EM Status Homed
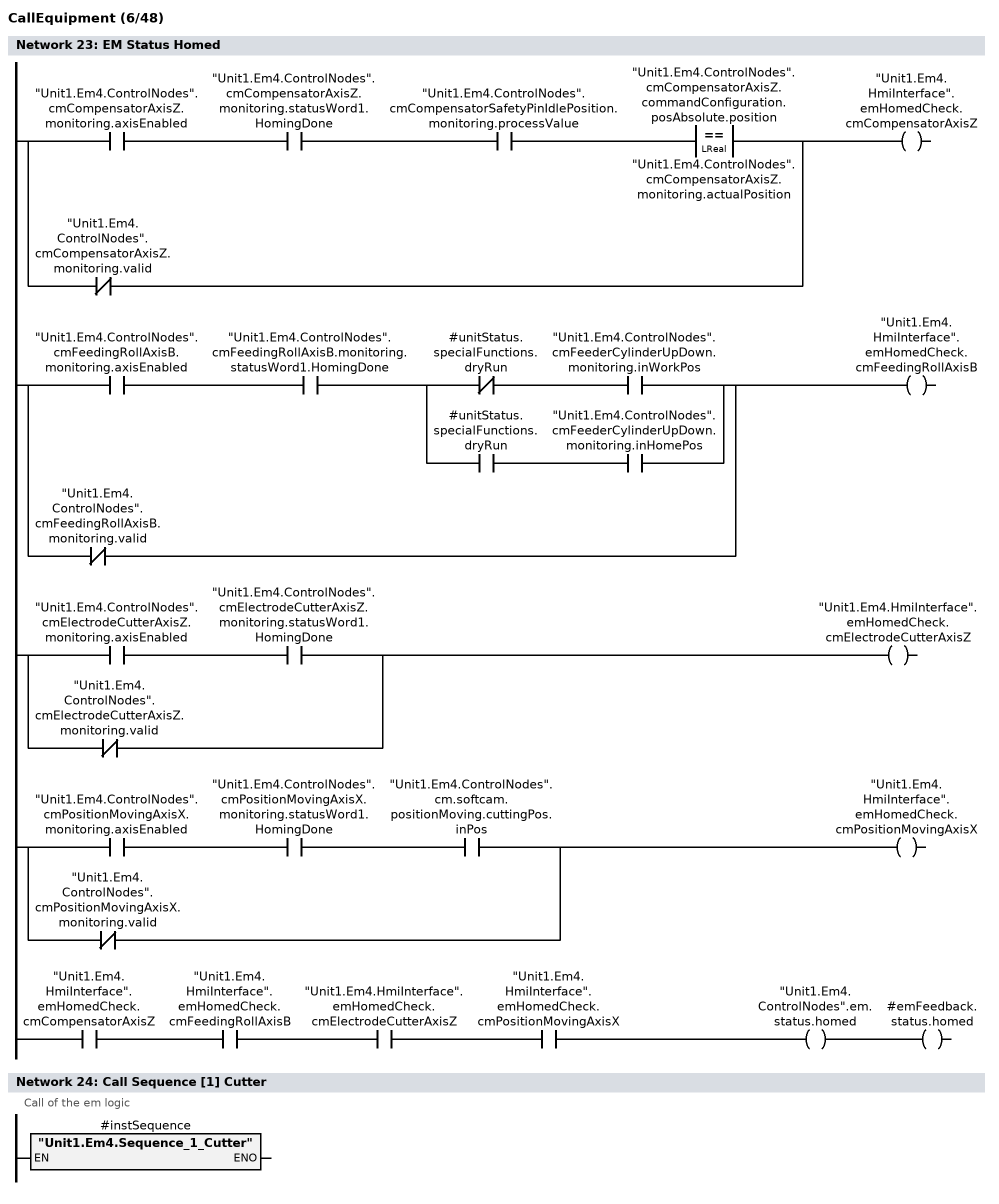
   RUNG wire#powerrail
      Contact( "Unit1.Em4.ControlNodes".cmCompensatorAxisZ.monitoring.axisEnabled )
      Contact( "Unit1.Em4.ControlNodes".cmCompensatorAxisZ.monitoring.statusWord1.HomingDone )
      Contact( "Unit1.Em4.ControlNodes".cmCompensatorSafetyPinIdlePosition.monitoring.processValue )
      { S7_Templates := "SrcType := LReal" } EQ_Contact(in1 := "Unit1.Em4.ControlNodes".cmCompensatorAxisZ.commandConfiguration.posAbsolute.position, in2 := "Unit1.Em4.ControlNodes".cmCompensatorAxisZ.monitoring.actualPosition)
      wire#w1
      Coil( "Unit1.Em4.HmiInterface".emHomedCheck.cmCompensatorAxisZ )
   END_RUNG
   RUNG wire#powerrail
      I_Contact( "Unit1.Em4.ControlNodes".cmCompensatorAxisZ.monitoring.valid )
   END_RUNG wire#w1
   RUNG wire#powerrail
      Contact( "Unit1.Em4.ControlNodes".cmFeedingRollAxisB.monitoring.axisEnabled )
      Contact( "Unit1.Em4.ControlNodes".cmFeedingRollAxisB.monitoring.statusWord1.HomingDone )
      wire#w2
      I_Contact( #unitStatus.specialFunctions.dryRun )
      Contact( "Unit1.Em4.ControlNodes".cmFeederCylinderUpDown.monitoring.inWorkPos )
      wire#w3
      Coil( "Unit1.Em4.HmiInterface".emHomedCheck.cmFeedingRollAxisB )
   END_RUNG
   RUNG wire#w2
      Contact( #unitStatus.specialFunctions.dryRun )
      Contact( "Unit1.Em4.ControlNodes".cmFeederCylinderUpDown.monitoring.inHomePos )
   END_RUNG wire#w3
   RUNG wire#powerrail
      I_Contact( "Unit1.Em4.ControlNodes".cmFeedingRollAxisB.monitoring.valid )
   END_RUNG wire#w3
   RUNG wire#powerrail
      Contact( "Unit1.Em4.ControlNodes".cmElectrodeCutterAxisZ.monitoring.axisEnabled )
      Contact( "Unit1.Em4.ControlNodes".cmElectrodeCutterAxisZ.monitoring.statusWord1.HomingDone )
      wire#w4
      Coil( "Unit1.Em4.HmiInterface".emHomedCheck.cmElectrodeCutterAxisZ )
   END_RUNG
   RUNG wire#powerrail
      I_Contact( "Unit1.Em4.ControlNodes".cmElectrodeCutterAxisZ.monitoring.valid )
   END_RUNG wire#w4
   RUNG wire#powerrail
      Contact( "Unit1.Em4.ControlNodes".cmPositionMovingAxisX.monitoring.axisEnabled )
      Contact( "Unit1.Em4.ControlNodes".cmPositionMovingAxisX.monitoring.statusWord1.HomingDone )
      Contact( "Unit1.Em4.ControlNodes".cm.softcam.positionMoving.cuttingPos.inPos )
      wire#w5
      Coil( "Unit1.Em4.HmiInterface".emHomedCheck.cmPositionMovingAxisX )
   END_RUNG
   RUNG wire#powerrail
      I_Contact( "Unit1.Em4.ControlNodes".cmPositionMovingAxisX.monitoring.valid )
   END_RUNG wire#w5
   RUNG wire#powerrail
      Contact( "Unit1.Em4.HmiInterface".emHomedCheck.cmCompensatorAxisZ )
      Contact( "Unit1.Em4.HmiInterface".emHomedCheck.cmFeedingRollAxisB )
      Contact( "Unit1.Em4.HmiInterface".emHomedCheck.cmElectrodeCutterAxisZ )
      Contact( "Unit1.Em4.HmiInterface".emHomedCheck.cmPositionMovingAxisX )
      Coil( "Unit1.Em4.ControlNodes".em.status.homed )
      Coil( #emFeedback.status.homed )
   END_RUNG
   // the same network as SCL:
   "Unit1.Em4.HmiInterface".emHomedCheck.cmCompensatorAxisZ := ("Unit1.Em4.ControlNodes".cmCompensatorAxisZ.monitoring.axisEnabled AND "Unit1.Em4.ControlNodes".cmCompensatorAxisZ.monitoring.statusWord1.HomingDone AND "Unit1.Em4.ControlNodes".cmCompensatorSafetyPinIdlePosition.monitoring.processValue AND ("Unit1.Em4.ControlNodes".cmCompensatorAxisZ.commandConfiguration.posAbsolute.position = "Unit1.Em4.ControlNodes".cmCompensatorAxisZ.monitoring.actualPosition)) OR NOT "Unit1.Em4.ControlNodes".cmCompensatorAxisZ.monitoring.valid;
   "Unit1.Em4.HmiInterface".emHomedCheck.cmFeedingRollAxisB := ("Unit1.Em4.ControlNodes".cmFeedingRollAxisB.monitoring.axisEnabled AND "Unit1.Em4.ControlNodes".cmFeedingRollAxisB.monitoring.statusWord1.HomingDone AND ((NOT #unitStatus.specialFunctions.dryRun AND "Unit1.Em4.ControlNodes".cmFeederCylinderUpDown.monitoring.inWorkPos) OR (#unitStatus.specialFunctions.dryRun AND "Unit1.Em4.ControlNodes".cmFeederCylinderUpDown.monitoring.inHomePos))) OR NOT "Unit1.Em4.ControlNodes".cmFeedingRollAxisB.monitoring.valid;
   "Unit1.Em4.HmiInterface".emHomedCheck.cmElectrodeCutterAxisZ := ("Unit1.Em4.ControlNodes".cmElectrodeCutterAxisZ.monitoring.axisEnabled AND "Unit1.Em4.ControlNodes".cmElectrodeCutterAxisZ.monitoring.statusWord1.HomingDone) OR NOT "Unit1.Em4.ControlNodes".cmElectrodeCutterAxisZ.monitoring.valid;
   "Unit1.Em4.HmiInterface".emHomedCheck.cmPositionMovingAxisX := ("Unit1.Em4.ControlNodes".cmPositionMovingAxisX.monitoring.axisEnabled AND "Unit1.Em4.ControlNodes".cmPositionMovingAxisX.monitoring.statusWord1.HomingDone AND "Unit1.Em4.ControlNodes".cm.softcam.positionMoving.cuttingPos.inPos) OR NOT "Unit1.Em4.ControlNodes".cmPositionMovingAxisX.monitoring.valid;
   "Unit1.Em4.ControlNodes".em.status.homed := "Unit1.Em4.HmiInterface".emHomedCheck.cmCompensatorAxisZ AND "Unit1.Em4.HmiInterface".emHomedCheck.cmFeedingRollAxisB AND "Unit1.Em4.HmiInterface".emHomedCheck.cmElectrodeCutterAxisZ AND "Unit1.Em4.HmiInterface".emHomedCheck.cmPositionMovingAxisX;
   #emFeedback.status.homed := "Unit1.Em4.ControlNodes".em.status.homed;
END_REGION

REGION Network 24: Call Sequence [1] Cutter
   // Call of the em logic
   RUNG wire#powerrail
      #instSequence()
   END_RUNG
   // the same network as SCL:
   #instSequence();   // "Unit1.Em4.Sequence_1_Cutter"
END_REGION

REGION Network 25: ******************** Part Data Generate ********************
END_REGION

REGION Network 27: ******************** Control Modules (Axis) ********************
   // Call control modules that are actuators after the em logic (jobs and sequence), so that the latest commands are applied to the actuators.
END_REGION

REGION Network 28: Reset CMS
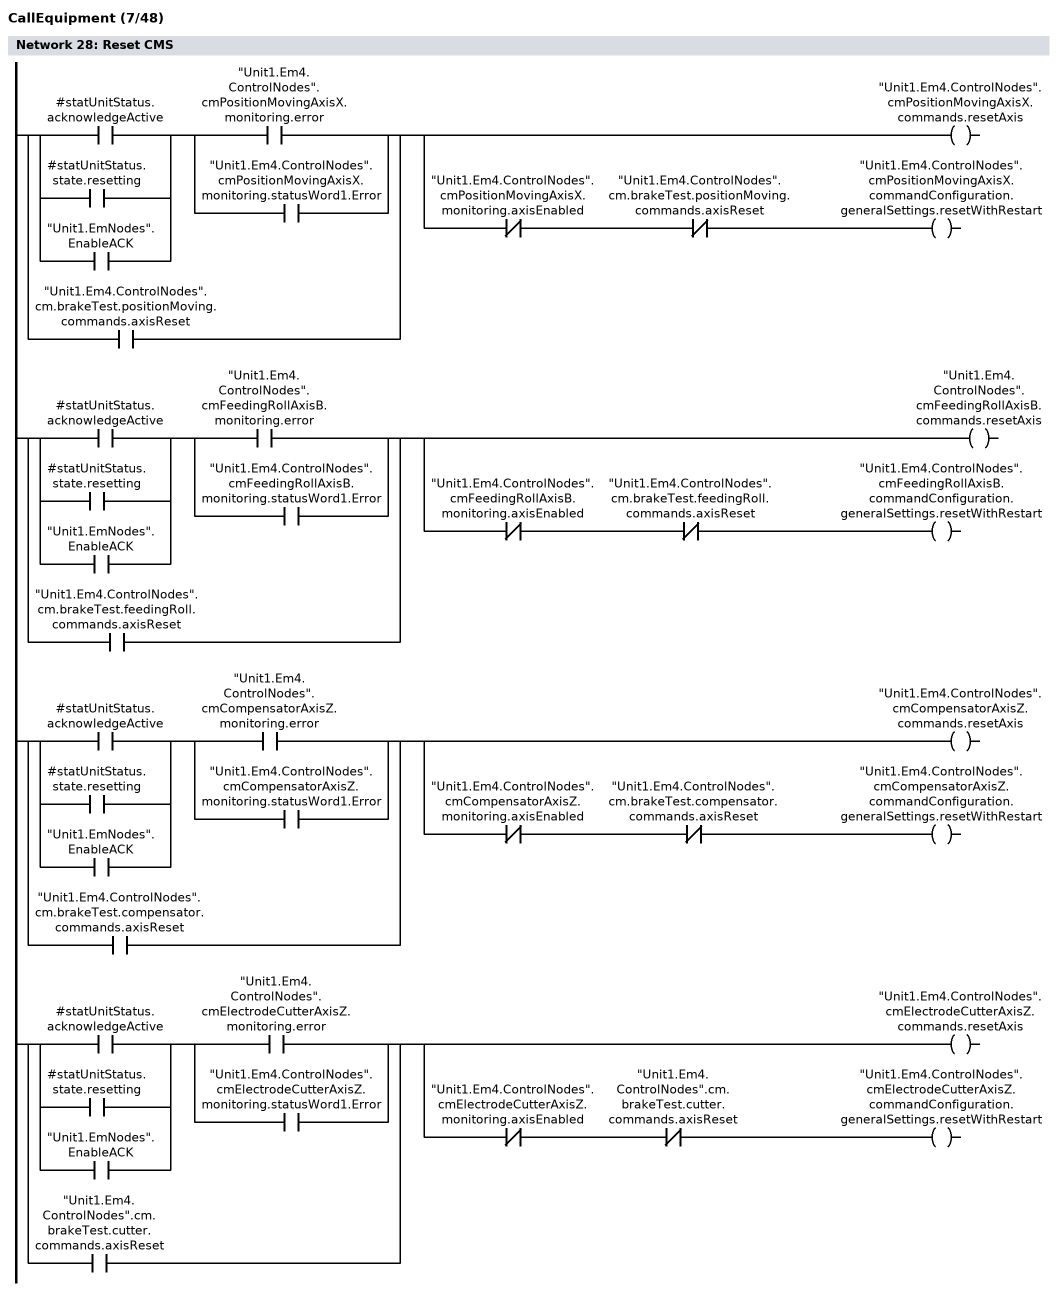
   RUNG wire#powerrail
      Contact( #statUnitStatus.acknowledgeActive )
      wire#w1
      Contact( "Unit1.Em4.ControlNodes".cmPositionMovingAxisX.monitoring.error )
      wire#w2
      Coil( "Unit1.Em4.ControlNodes".cmPositionMovingAxisX.commands.resetAxis )
   END_RUNG
   RUNG wire#powerrail
      Contact( #statUnitStatus.state.resetting )
   END_RUNG wire#w1
   RUNG wire#powerrail
      Contact( "Unit1.EmNodes".EnableACK )
   END_RUNG wire#w1
   RUNG wire#w1
      Contact( "Unit1.Em4.ControlNodes".cmPositionMovingAxisX.monitoring.statusWord1.Error )
   END_RUNG wire#w2
   RUNG wire#powerrail
      Contact( "Unit1.Em4.ControlNodes".cm.brakeTest.positionMoving.commands.axisReset )
   END_RUNG wire#w2
   RUNG wire#w2
      I_Contact( "Unit1.Em4.ControlNodes".cmPositionMovingAxisX.monitoring.axisEnabled )
      I_Contact( "Unit1.Em4.ControlNodes".cm.brakeTest.positionMoving.commands.axisReset )
      Coil( "Unit1.Em4.ControlNodes".cmPositionMovingAxisX.commandConfiguration.generalSettings.resetWithRestart )
   END_RUNG
   RUNG wire#powerrail
      Contact( #statUnitStatus.acknowledgeActive )
      wire#w3
      Contact( "Unit1.Em4.ControlNodes".cmFeedingRollAxisB.monitoring.error )
      wire#w4
      Coil( "Unit1.Em4.ControlNodes".cmFeedingRollAxisB.commands.resetAxis )
   END_RUNG
   RUNG wire#powerrail
      Contact( #statUnitStatus.state.resetting )
   END_RUNG wire#w3
   RUNG wire#powerrail
      Contact( "Unit1.EmNodes".EnableACK )
   END_RUNG wire#w3
   RUNG wire#w3
      Contact( "Unit1.Em4.ControlNodes".cmFeedingRollAxisB.monitoring.statusWord1.Error )
   END_RUNG wire#w4
   RUNG wire#powerrail
      Contact( "Unit1.Em4.ControlNodes".cm.brakeTest.feedingRoll.commands.axisReset )
   END_RUNG wire#w4
   RUNG wire#w4
      I_Contact( "Unit1.Em4.ControlNodes".cmFeedingRollAxisB.monitoring.axisEnabled )
      I_Contact( "Unit1.Em4.ControlNodes".cm.brakeTest.feedingRoll.commands.axisReset )
      Coil( "Unit1.Em4.ControlNodes".cmFeedingRollAxisB.commandConfiguration.generalSettings.resetWithRestart )
   END_RUNG
   RUNG wire#powerrail
      Contact( #statUnitStatus.acknowledgeActive )
      wire#w5
      Contact( "Unit1.Em4.ControlNodes".cmCompensatorAxisZ.monitoring.error )
      wire#w6
      Coil( "Unit1.Em4.ControlNodes".cmCompensatorAxisZ.commands.resetAxis )
   END_RUNG
   RUNG wire#powerrail
      Contact( #statUnitStatus.state.resetting )
   END_RUNG wire#w5
   RUNG wire#powerrail
      Contact( "Unit1.EmNodes".EnableACK )
   END_RUNG wire#w5
   RUNG wire#w5
      Contact( "Unit1.Em4.ControlNodes".cmCompensatorAxisZ.monitoring.statusWord1.Error )
   END_RUNG wire#w6
   RUNG wire#powerrail
      Contact( "Unit1.Em4.ControlNodes".cm.brakeTest.compensator.commands.axisReset )
   END_RUNG wire#w6
   RUNG wire#w6
      I_Contact( "Unit1.Em4.ControlNodes".cmCompensatorAxisZ.monitoring.axisEnabled )
      I_Contact( "Unit1.Em4.ControlNodes".cm.brakeTest.compensator.commands.axisReset )
      Coil( "Unit1.Em4.ControlNodes".cmCompensatorAxisZ.commandConfiguration.generalSettings.resetWithRestart )
   END_RUNG
   RUNG wire#powerrail
      Contact( #statUnitStatus.acknowledgeActive )
      wire#w7
      Contact( "Unit1.Em4.ControlNodes".cmElectrodeCutterAxisZ.monitoring.error )
      wire#w8
      Coil( "Unit1.Em4.ControlNodes".cmElectrodeCutterAxisZ.commands.resetAxis )
   END_RUNG
   RUNG wire#powerrail
      Contact( #statUnitStatus.state.resetting )
   END_RUNG wire#w7
   RUNG wire#powerrail
      Contact( "Unit1.EmNodes".EnableACK )
   END_RUNG wire#w7
   RUNG wire#w7
      Contact( "Unit1.Em4.ControlNodes".cmElectrodeCutterAxisZ.monitoring.statusWord1.Error )
   END_RUNG wire#w8
   RUNG wire#powerrail
      Contact( "Unit1.Em4.ControlNodes".cm.brakeTest.cutter.commands.axisReset )
   END_RUNG wire#w8
   RUNG wire#w8
      I_Contact( "Unit1.Em4.ControlNodes".cmElectrodeCutterAxisZ.monitoring.axisEnabled )
      I_Contact( "Unit1.Em4.ControlNodes".cm.brakeTest.cutter.commands.axisReset )
      Coil( "Unit1.Em4.ControlNodes".cmElectrodeCutterAxisZ.commandConfiguration.generalSettings.resetWithRestart )
   END_RUNG
   // the same network as SCL:
   "Unit1.Em4.ControlNodes".cmPositionMovingAxisX.commands.resetAxis := ((#statUnitStatus.acknowledgeActive OR #statUnitStatus.state.resetting OR "Unit1.EmNodes".EnableACK) AND ("Unit1.Em4.ControlNodes".cmPositionMovingAxisX.monitoring.error OR "Unit1.Em4.ControlNodes".cmPositionMovingAxisX.monitoring.statusWord1.Error)) OR "Unit1.Em4.ControlNodes".cm.brakeTest.positionMoving.commands.axisReset;
   "Unit1.Em4.ControlNodes".cmPositionMovingAxisX.commandConfiguration.generalSettings.resetWithRestart := "Unit1.Em4.ControlNodes".cmPositionMovingAxisX.commands.resetAxis AND NOT "Unit1.Em4.ControlNodes".cmPositionMovingAxisX.monitoring.axisEnabled AND NOT "Unit1.Em4.ControlNodes".cm.brakeTest.positionMoving.commands.axisReset;
   "Unit1.Em4.ControlNodes".cmFeedingRollAxisB.commands.resetAxis := ((#statUnitStatus.acknowledgeActive OR #statUnitStatus.state.resetting OR "Unit1.EmNodes".EnableACK) AND ("Unit1.Em4.ControlNodes".cmFeedingRollAxisB.monitoring.error OR "Unit1.Em4.ControlNodes".cmFeedingRollAxisB.monitoring.statusWord1.Error)) OR "Unit1.Em4.ControlNodes".cm.brakeTest.feedingRoll.commands.axisReset;
   "Unit1.Em4.ControlNodes".cmFeedingRollAxisB.commandConfiguration.generalSettings.resetWithRestart := "Unit1.Em4.ControlNodes".cmFeedingRollAxisB.commands.resetAxis AND NOT "Unit1.Em4.ControlNodes".cmFeedingRollAxisB.monitoring.axisEnabled AND NOT "Unit1.Em4.ControlNodes".cm.brakeTest.feedingRoll.commands.axisReset;
   "Unit1.Em4.ControlNodes".cmCompensatorAxisZ.commands.resetAxis := ((#statUnitStatus.acknowledgeActive OR #statUnitStatus.state.resetting OR "Unit1.EmNodes".EnableACK) AND ("Unit1.Em4.ControlNodes".cmCompensatorAxisZ.monitoring.error OR "Unit1.Em4.ControlNodes".cmCompensatorAxisZ.monitoring.statusWord1.Error)) OR "Unit1.Em4.ControlNodes".cm.brakeTest.compensator.commands.axisReset;
   "Unit1.Em4.ControlNodes".cmCompensatorAxisZ.commandConfiguration.generalSettings.resetWithRestart := "Unit1.Em4.ControlNodes".cmCompensatorAxisZ.commands.resetAxis AND NOT "Unit1.Em4.ControlNodes".cmCompensatorAxisZ.monitoring.axisEnabled AND NOT "Unit1.Em4.ControlNodes".cm.brakeTest.compensator.commands.axisReset;
   "Unit1.Em4.ControlNodes".cmElectrodeCutterAxisZ.commands.resetAxis := ((#statUnitStatus.acknowledgeActive OR #statUnitStatus.state.resetting OR "Unit1.EmNodes".EnableACK) AND ("Unit1.Em4.ControlNodes".cmElectrodeCutterAxisZ.monitoring.error OR "Unit1.Em4.ControlNodes".cmElectrodeCutterAxisZ.monitoring.statusWord1.Error)) OR "Unit1.Em4.ControlNodes".cm.brakeTest.cutter.commands.axisReset;
   "Unit1.Em4.ControlNodes".cmElectrodeCutterAxisZ.commandConfiguration.generalSettings.resetWithRestart := "Unit1.Em4.ControlNodes".cmElectrodeCutterAxisZ.commands.resetAxis AND NOT "Unit1.Em4.ControlNodes".cmElectrodeCutterAxisZ.monitoring.axisEnabled AND NOT "Unit1.Em4.ControlNodes".cm.brakeTest.cutter.commands.axisReset;
END_REGION

REGION Network 29: Enable/Disable CMs
   // Enable the axis during the resetting state and disable the axis during the aborting state.
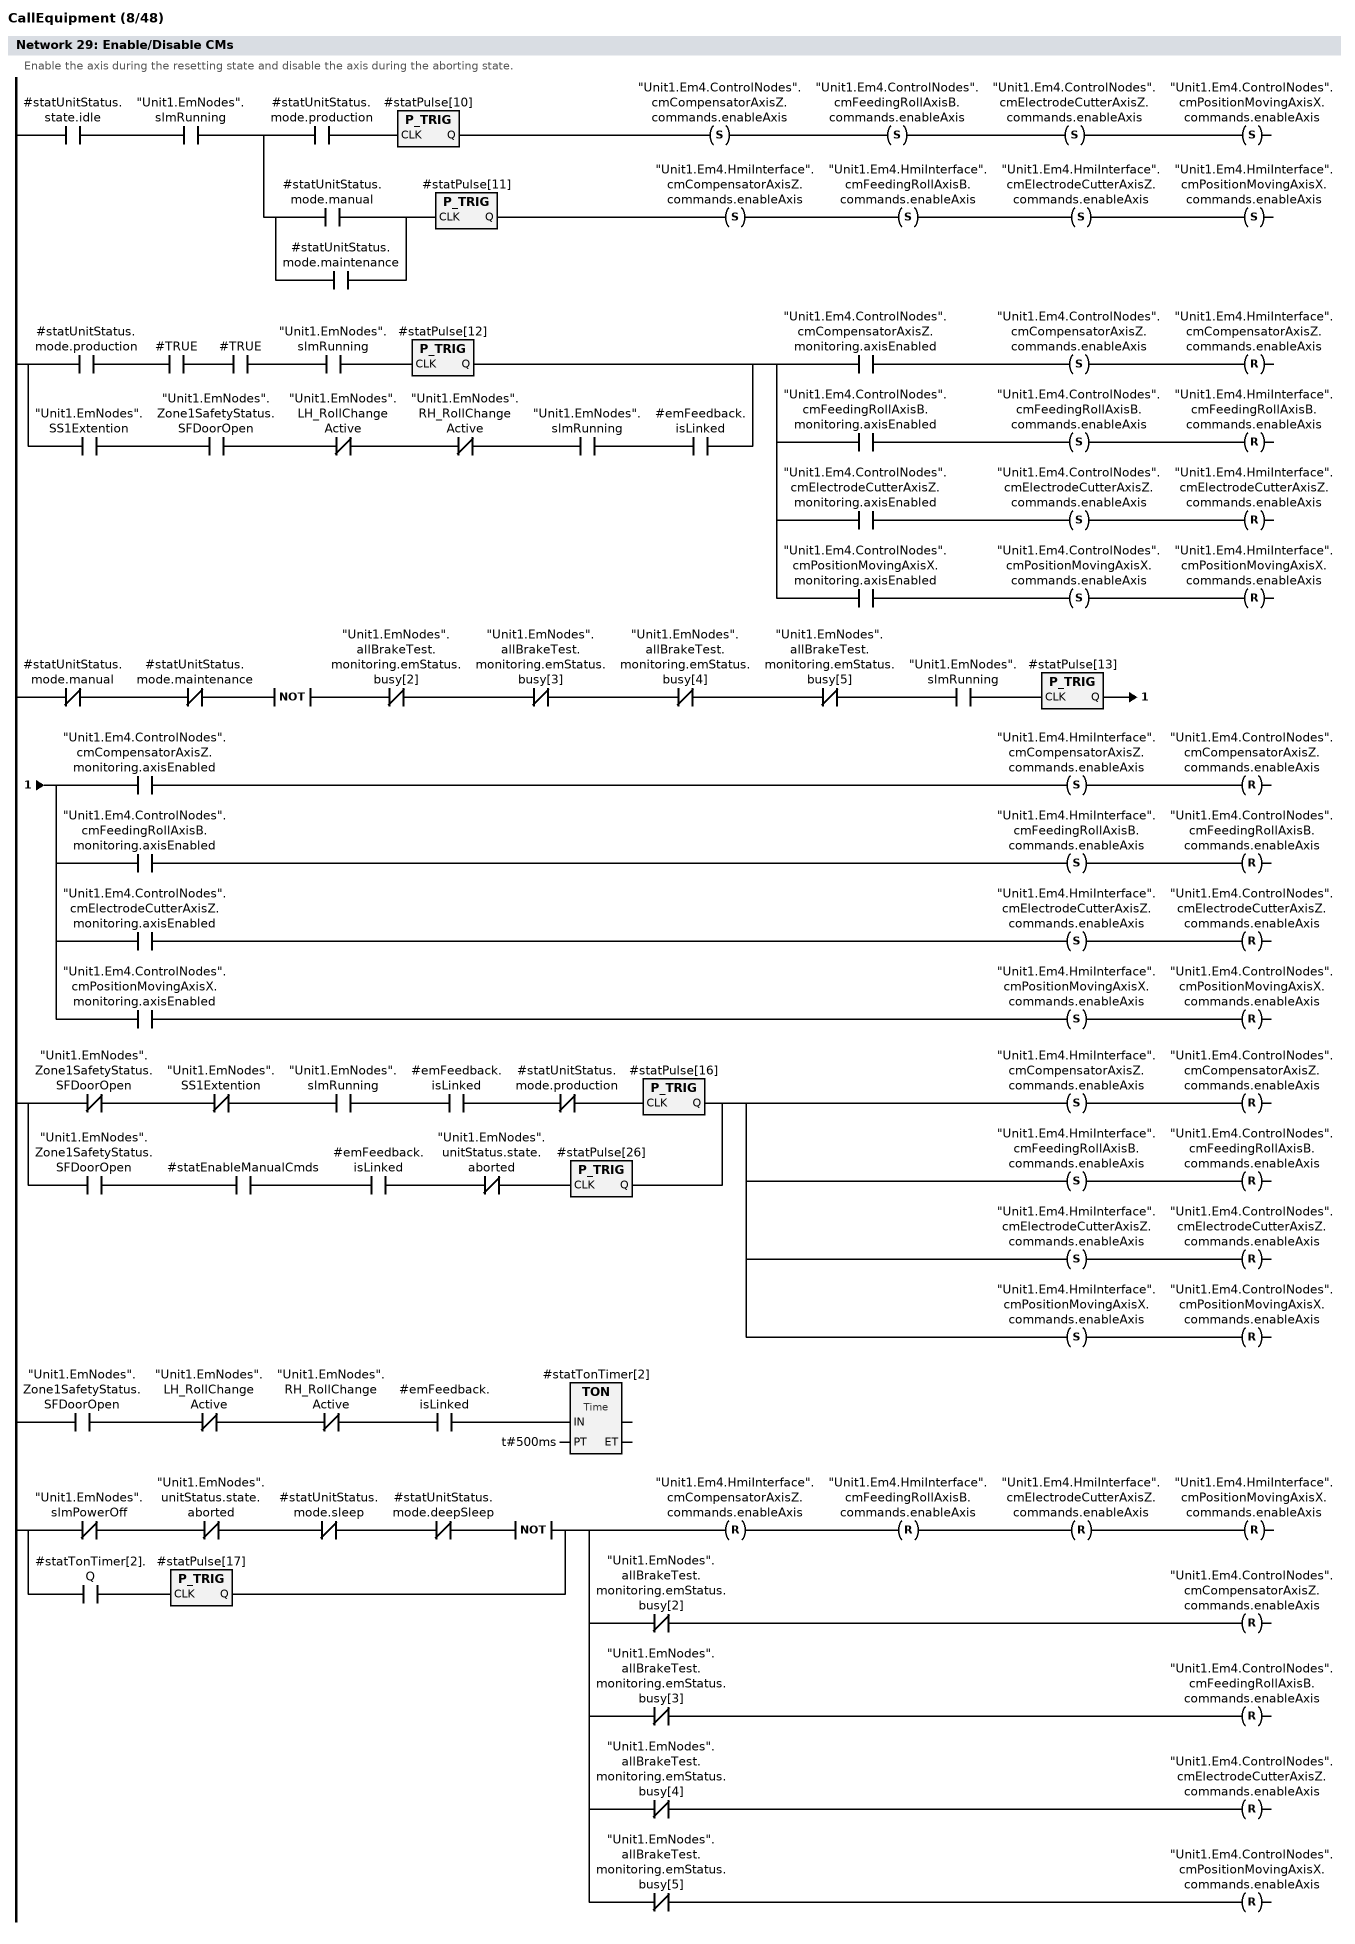
   RUNG wire#powerrail
      Contact( #statUnitStatus.state.idle )
      Contact( "Unit1.EmNodes".slmRunning )
      wire#w1
      Contact( #statUnitStatus.mode.production )
      P_Trig( #statPulse[10] )
      S_Coil( "Unit1.Em4.ControlNodes".cmCompensatorAxisZ.commands.enableAxis )
      S_Coil( "Unit1.Em4.ControlNodes".cmFeedingRollAxisB.commands.enableAxis )
      S_Coil( "Unit1.Em4.ControlNodes".cmElectrodeCutterAxisZ.commands.enableAxis )
      S_Coil( "Unit1.Em4.ControlNodes".cmPositionMovingAxisX.commands.enableAxis )
   END_RUNG
   RUNG wire#w1
      Contact( #statUnitStatus.mode.manual )
      wire#w2
      P_Trig( #statPulse[11] )
      S_Coil( "Unit1.Em4.HmiInterface".cmCompensatorAxisZ.commands.enableAxis )
      S_Coil( "Unit1.Em4.HmiInterface".cmFeedingRollAxisB.commands.enableAxis )
      S_Coil( "Unit1.Em4.HmiInterface".cmElectrodeCutterAxisZ.commands.enableAxis )
      S_Coil( "Unit1.Em4.HmiInterface".cmPositionMovingAxisX.commands.enableAxis )
   END_RUNG
   RUNG wire#w1
      Contact( #statUnitStatus.mode.maintenance )
   END_RUNG wire#w2
   RUNG wire#powerrail
      Contact( #statUnitStatus.mode.production )
      Contact( #TRUE )
      Contact( #TRUE )
      Contact( "Unit1.EmNodes".slmRunning )
      P_Trig( #statPulse[12] )
      wire#w3
      Contact( "Unit1.Em4.ControlNodes".cmCompensatorAxisZ.monitoring.axisEnabled )
      S_Coil( "Unit1.Em4.ControlNodes".cmCompensatorAxisZ.commands.enableAxis )
      R_Coil( "Unit1.Em4.HmiInterface".cmCompensatorAxisZ.commands.enableAxis )
   END_RUNG
   RUNG wire#powerrail
      Contact( "Unit1.EmNodes".SS1Extention )
      Contact( "Unit1.EmNodes".Zone1SafetyStatus.SFDoorOpen )
      I_Contact( "Unit1.EmNodes".LH_RollChangeActive )
      I_Contact( "Unit1.EmNodes".RH_RollChangeActive )
      Contact( "Unit1.EmNodes".slmRunning )
      Contact( #emFeedback.isLinked )
   END_RUNG wire#w3
   RUNG wire#w3
      Contact( "Unit1.Em4.ControlNodes".cmFeedingRollAxisB.monitoring.axisEnabled )
      S_Coil( "Unit1.Em4.ControlNodes".cmFeedingRollAxisB.commands.enableAxis )
      R_Coil( "Unit1.Em4.HmiInterface".cmFeedingRollAxisB.commands.enableAxis )
   END_RUNG
   RUNG wire#w3
      Contact( "Unit1.Em4.ControlNodes".cmElectrodeCutterAxisZ.monitoring.axisEnabled )
      S_Coil( "Unit1.Em4.ControlNodes".cmElectrodeCutterAxisZ.commands.enableAxis )
      R_Coil( "Unit1.Em4.HmiInterface".cmElectrodeCutterAxisZ.commands.enableAxis )
   END_RUNG
   RUNG wire#w3
      Contact( "Unit1.Em4.ControlNodes".cmPositionMovingAxisX.monitoring.axisEnabled )
      S_Coil( "Unit1.Em4.ControlNodes".cmPositionMovingAxisX.commands.enableAxis )
      R_Coil( "Unit1.Em4.HmiInterface".cmPositionMovingAxisX.commands.enableAxis )
   END_RUNG
   RUNG wire#powerrail
      I_Contact( #statUnitStatus.mode.manual )
      I_Contact( #statUnitStatus.mode.maintenance )
      Not()
      I_Contact( "Unit1.EmNodes".allBrakeTest.monitoring.emStatus.busy[2] )
      I_Contact( "Unit1.EmNodes".allBrakeTest.monitoring.emStatus.busy[3] )
      I_Contact( "Unit1.EmNodes".allBrakeTest.monitoring.emStatus.busy[4] )
      I_Contact( "Unit1.EmNodes".allBrakeTest.monitoring.emStatus.busy[5] )
      Contact( "Unit1.EmNodes".slmRunning )
      P_Trig( #statPulse[13] )
      wire#w4
      Contact( "Unit1.Em4.ControlNodes".cmCompensatorAxisZ.monitoring.axisEnabled )
      S_Coil( "Unit1.Em4.HmiInterface".cmCompensatorAxisZ.commands.enableAxis )
      R_Coil( "Unit1.Em4.ControlNodes".cmCompensatorAxisZ.commands.enableAxis )
   END_RUNG
   RUNG wire#w4
      Contact( "Unit1.Em4.ControlNodes".cmFeedingRollAxisB.monitoring.axisEnabled )
      S_Coil( "Unit1.Em4.HmiInterface".cmFeedingRollAxisB.commands.enableAxis )
      R_Coil( "Unit1.Em4.ControlNodes".cmFeedingRollAxisB.commands.enableAxis )
   END_RUNG
   RUNG wire#w4
      Contact( "Unit1.Em4.ControlNodes".cmElectrodeCutterAxisZ.monitoring.axisEnabled )
      S_Coil( "Unit1.Em4.HmiInterface".cmElectrodeCutterAxisZ.commands.enableAxis )
      R_Coil( "Unit1.Em4.ControlNodes".cmElectrodeCutterAxisZ.commands.enableAxis )
   END_RUNG
   RUNG wire#w4
      Contact( "Unit1.Em4.ControlNodes".cmPositionMovingAxisX.monitoring.axisEnabled )
      S_Coil( "Unit1.Em4.HmiInterface".cmPositionMovingAxisX.commands.enableAxis )
      R_Coil( "Unit1.Em4.ControlNodes".cmPositionMovingAxisX.commands.enableAxis )
   END_RUNG
   RUNG wire#powerrail
      I_Contact( "Unit1.EmNodes".Zone1SafetyStatus.SFDoorOpen )
      I_Contact( "Unit1.EmNodes".SS1Extention )
      Contact( "Unit1.EmNodes".slmRunning )
      Contact( #emFeedback.isLinked )
      I_Contact( #statUnitStatus.mode.production )
      P_Trig( #statPulse[16] )
      wire#w5
      S_Coil( "Unit1.Em4.HmiInterface".cmCompensatorAxisZ.commands.enableAxis )
      R_Coil( "Unit1.Em4.ControlNodes".cmCompensatorAxisZ.commands.enableAxis )
   END_RUNG
   RUNG wire#powerrail
      Contact( "Unit1.EmNodes".Zone1SafetyStatus.SFDoorOpen )
      Contact( #statEnableManualCmds )
      Contact( #emFeedback.isLinked )
      I_Contact( "Unit1.EmNodes".unitStatus.state.aborted )
      P_Trig( #statPulse[26] )
   END_RUNG wire#w5
   RUNG wire#w5
      S_Coil( "Unit1.Em4.HmiInterface".cmFeedingRollAxisB.commands.enableAxis )
      R_Coil( "Unit1.Em4.ControlNodes".cmFeedingRollAxisB.commands.enableAxis )
   END_RUNG
   RUNG wire#w5
      S_Coil( "Unit1.Em4.HmiInterface".cmElectrodeCutterAxisZ.commands.enableAxis )
      R_Coil( "Unit1.Em4.ControlNodes".cmElectrodeCutterAxisZ.commands.enableAxis )
   END_RUNG
   RUNG wire#w5
      S_Coil( "Unit1.Em4.HmiInterface".cmPositionMovingAxisX.commands.enableAxis )
      R_Coil( "Unit1.Em4.ControlNodes".cmPositionMovingAxisX.commands.enableAxis )
   END_RUNG
   RUNG wire#powerrail
      Contact( "Unit1.EmNodes".Zone1SafetyStatus.SFDoorOpen )
      I_Contact( "Unit1.EmNodes".LH_RollChangeActive )
      I_Contact( "Unit1.EmNodes".RH_RollChangeActive )
      Contact( #emFeedback.isLinked )
      { S7_Templates := "time_type := Time" } #statTonTimer[2].TON(pt := t#500ms, et =>)
   END_RUNG
   RUNG wire#powerrail
      I_Contact( "Unit1.EmNodes".slmPowerOff )
      I_Contact( "Unit1.EmNodes".unitStatus.state.aborted )
      I_Contact( #statUnitStatus.mode.sleep )
      I_Contact( #statUnitStatus.mode.deepSleep )
      Not()
      wire#w6
      R_Coil( "Unit1.Em4.HmiInterface".cmCompensatorAxisZ.commands.enableAxis )
      R_Coil( "Unit1.Em4.HmiInterface".cmFeedingRollAxisB.commands.enableAxis )
      R_Coil( "Unit1.Em4.HmiInterface".cmElectrodeCutterAxisZ.commands.enableAxis )
      R_Coil( "Unit1.Em4.HmiInterface".cmPositionMovingAxisX.commands.enableAxis )
   END_RUNG
   RUNG wire#powerrail
      Contact( #statTonTimer[2].Q )
      P_Trig( #statPulse[17] )
   END_RUNG wire#w6
   RUNG wire#w6
      I_Contact( "Unit1.EmNodes".allBrakeTest.monitoring.emStatus.busy[2] )
      R_Coil( "Unit1.Em4.ControlNodes".cmCompensatorAxisZ.commands.enableAxis )
   END_RUNG
   RUNG wire#w6
      I_Contact( "Unit1.EmNodes".allBrakeTest.monitoring.emStatus.busy[3] )
      R_Coil( "Unit1.Em4.ControlNodes".cmFeedingRollAxisB.commands.enableAxis )
   END_RUNG
   RUNG wire#w6
      I_Contact( "Unit1.EmNodes".allBrakeTest.monitoring.emStatus.busy[4] )
      R_Coil( "Unit1.Em4.ControlNodes".cmElectrodeCutterAxisZ.commands.enableAxis )
   END_RUNG
   RUNG wire#w6
      I_Contact( "Unit1.EmNodes".allBrakeTest.monitoring.emStatus.busy[5] )
      R_Coil( "Unit1.Em4.ControlNodes".cmPositionMovingAxisX.commands.enableAxis )
   END_RUNG
   // the same network as SCL:
   #_w1 := #statUnitStatus.state.idle AND "Unit1.EmNodes".slmRunning;
   #_w2 := #_w1 AND #statUnitStatus.mode.production;
   #_w3 := #_w2 AND NOT #statPulse[10];   // rising edge
   #statPulse[10] := #_w2;
   IF #_w3 THEN
       "Unit1.Em4.ControlNodes".cmCompensatorAxisZ.commands.enableAxis := TRUE;
       "Unit1.Em4.ControlNodes".cmFeedingRollAxisB.commands.enableAxis := TRUE;
       "Unit1.Em4.ControlNodes".cmElectrodeCutterAxisZ.commands.enableAxis := TRUE;
       "Unit1.Em4.ControlNodes".cmPositionMovingAxisX.commands.enableAxis := TRUE;
   END_IF;
   #_w4 := #_w1 AND (#statUnitStatus.mode.manual OR #statUnitStatus.mode.maintenance);
   #_w5 := #_w4 AND NOT #statPulse[11];   // rising edge
   #statPulse[11] := #_w4;
   IF #_w5 THEN
       "Unit1.Em4.HmiInterface".cmCompensatorAxisZ.commands.enableAxis := TRUE;
       "Unit1.Em4.HmiInterface".cmFeedingRollAxisB.commands.enableAxis := TRUE;
       "Unit1.Em4.HmiInterface".cmElectrodeCutterAxisZ.commands.enableAxis := TRUE;
       "Unit1.Em4.HmiInterface".cmPositionMovingAxisX.commands.enableAxis := TRUE;
   END_IF;
   #_w6 := #statUnitStatus.mode.production AND #TRUE AND #TRUE AND "Unit1.EmNodes".slmRunning;
   #_w7 := #_w6 AND NOT #statPulse[12];   // rising edge
   #statPulse[12] := #_w6;
   #_w8 := #_w7 OR ("Unit1.EmNodes".SS1Extention AND "Unit1.EmNodes".Zone1SafetyStatus.SFDoorOpen AND NOT "Unit1.EmNodes".LH_RollChangeActive AND NOT "Unit1.EmNodes".RH_RollChangeActive AND "Unit1.EmNodes".slmRunning AND #emFeedback.isLinked);
   IF #_w8 AND "Unit1.Em4.ControlNodes".cmCompensatorAxisZ.monitoring.axisEnabled THEN
       "Unit1.Em4.ControlNodes".cmCompensatorAxisZ.commands.enableAxis := TRUE;
       "Unit1.Em4.HmiInterface".cmCompensatorAxisZ.commands.enableAxis := FALSE;
   END_IF;
   IF #_w8 AND "Unit1.Em4.ControlNodes".cmFeedingRollAxisB.monitoring.axisEnabled THEN
       "Unit1.Em4.ControlNodes".cmFeedingRollAxisB.commands.enableAxis := TRUE;
       "Unit1.Em4.HmiInterface".cmFeedingRollAxisB.commands.enableAxis := FALSE;
   END_IF;
   IF #_w8 AND "Unit1.Em4.ControlNodes".cmElectrodeCutterAxisZ.monitoring.axisEnabled THEN
       "Unit1.Em4.ControlNodes".cmElectrodeCutterAxisZ.commands.enableAxis := TRUE;
       "Unit1.Em4.HmiInterface".cmElectrodeCutterAxisZ.commands.enableAxis := FALSE;
   END_IF;
   IF #_w8 AND "Unit1.Em4.ControlNodes".cmPositionMovingAxisX.monitoring.axisEnabled THEN
       "Unit1.Em4.ControlNodes".cmPositionMovingAxisX.commands.enableAxis := TRUE;
       "Unit1.Em4.HmiInterface".cmPositionMovingAxisX.commands.enableAxis := FALSE;
   END_IF;
   #_w9 := NOT (NOT #statUnitStatus.mode.manual AND NOT #statUnitStatus.mode.maintenance) AND NOT "Unit1.EmNodes".allBrakeTest.monitoring.emStatus.busy[2] AND NOT "Unit1.EmNodes".allBrakeTest.monitoring.emStatus.busy[3] AND NOT "Unit1.EmNodes".allBrakeTest.monitoring.emStatus.busy[4] AND NOT "Unit1.EmNodes".allBrakeTest.monitoring.emStatus.busy[5] AND "Unit1.EmNodes".slmRunning;
   #_w10 := #_w9 AND NOT #statPulse[13];   // rising edge
   #statPulse[13] := #_w9;
   IF #_w10 AND "Unit1.Em4.ControlNodes".cmCompensatorAxisZ.monitoring.axisEnabled THEN
       "Unit1.Em4.HmiInterface".cmCompensatorAxisZ.commands.enableAxis := TRUE;
       "Unit1.Em4.ControlNodes".cmCompensatorAxisZ.commands.enableAxis := FALSE;
   END_IF;
   IF #_w10 AND "Unit1.Em4.ControlNodes".cmFeedingRollAxisB.monitoring.axisEnabled THEN
       "Unit1.Em4.HmiInterface".cmFeedingRollAxisB.commands.enableAxis := TRUE;
       "Unit1.Em4.ControlNodes".cmFeedingRollAxisB.commands.enableAxis := FALSE;
   END_IF;
   IF #_w10 AND "Unit1.Em4.ControlNodes".cmElectrodeCutterAxisZ.monitoring.axisEnabled THEN
       "Unit1.Em4.HmiInterface".cmElectrodeCutterAxisZ.commands.enableAxis := TRUE;
       "Unit1.Em4.ControlNodes".cmElectrodeCutterAxisZ.commands.enableAxis := FALSE;
   END_IF;
   IF #_w10 AND "Unit1.Em4.ControlNodes".cmPositionMovingAxisX.monitoring.axisEnabled THEN
       "Unit1.Em4.HmiInterface".cmPositionMovingAxisX.commands.enableAxis := TRUE;
       "Unit1.Em4.ControlNodes".cmPositionMovingAxisX.commands.enableAxis := FALSE;
   END_IF;
   #_w11 := NOT "Unit1.EmNodes".Zone1SafetyStatus.SFDoorOpen AND NOT "Unit1.EmNodes".SS1Extention AND "Unit1.EmNodes".slmRunning AND #emFeedback.isLinked AND NOT #statUnitStatus.mode.production;
   #_w12 := #_w11 AND NOT #statPulse[16];   // rising edge
   #statPulse[16] := #_w11;
   #_w13 := "Unit1.EmNodes".Zone1SafetyStatus.SFDoorOpen AND #statEnableManualCmds AND #emFeedback.isLinked AND NOT "Unit1.EmNodes".unitStatus.state.aborted;
   #_w14 := #_w13 AND NOT #statPulse[26];   // rising edge
   #statPulse[26] := #_w13;
   IF #_w12 OR #_w14 THEN
       "Unit1.Em4.HmiInterface".cmCompensatorAxisZ.commands.enableAxis := TRUE;
       "Unit1.Em4.ControlNodes".cmCompensatorAxisZ.commands.enableAxis := FALSE;
       "Unit1.Em4.HmiInterface".cmFeedingRollAxisB.commands.enableAxis := TRUE;
       "Unit1.Em4.ControlNodes".cmFeedingRollAxisB.commands.enableAxis := FALSE;
       "Unit1.Em4.HmiInterface".cmElectrodeCutterAxisZ.commands.enableAxis := TRUE;
       "Unit1.Em4.ControlNodes".cmElectrodeCutterAxisZ.commands.enableAxis := FALSE;
       "Unit1.Em4.HmiInterface".cmPositionMovingAxisX.commands.enableAxis := TRUE;
       "Unit1.Em4.ControlNodes".cmPositionMovingAxisX.commands.enableAxis := FALSE;
   END_IF;
   #statTonTimer[2].TON(IN := "Unit1.EmNodes".Zone1SafetyStatus.SFDoorOpen AND NOT "Unit1.EmNodes".LH_RollChangeActive AND NOT "Unit1.EmNodes".RH_RollChangeActive AND #emFeedback.isLinked,
                        PT := t#500ms);
   #_w15 := #statTonTimer[2].Q AND NOT #statPulse[17];   // rising edge
   #statPulse[17] := #statTonTimer[2].Q;
   #_w16 := NOT (NOT "Unit1.EmNodes".slmPowerOff AND NOT "Unit1.EmNodes".unitStatus.state.aborted AND NOT #statUnitStatus.mode.sleep AND NOT #statUnitStatus.mode.deepSleep) OR #_w15;
   IF #_w16 THEN
       "Unit1.Em4.HmiInterface".cmCompensatorAxisZ.commands.enableAxis := FALSE;
       "Unit1.Em4.HmiInterface".cmFeedingRollAxisB.commands.enableAxis := FALSE;
       "Unit1.Em4.HmiInterface".cmElectrodeCutterAxisZ.commands.enableAxis := FALSE;
       "Unit1.Em4.HmiInterface".cmPositionMovingAxisX.commands.enableAxis := FALSE;
   END_IF;
   IF #_w16 AND NOT "Unit1.EmNodes".allBrakeTest.monitoring.emStatus.busy[2] THEN
       "Unit1.Em4.ControlNodes".cmCompensatorAxisZ.commands.enableAxis := FALSE;
   END_IF;
   IF #_w16 AND NOT "Unit1.EmNodes".allBrakeTest.monitoring.emStatus.busy[3] THEN
       "Unit1.Em4.ControlNodes".cmFeedingRollAxisB.commands.enableAxis := FALSE;
   END_IF;
   IF #_w16 AND NOT "Unit1.EmNodes".allBrakeTest.monitoring.emStatus.busy[4] THEN
       "Unit1.Em4.ControlNodes".cmElectrodeCutterAxisZ.commands.enableAxis := FALSE;
   END_IF;
   IF #_w16 AND NOT "Unit1.EmNodes".allBrakeTest.monitoring.emStatus.busy[5] THEN
       "Unit1.Em4.ControlNodes".cmPositionMovingAxisX.commands.enableAxis := FALSE;
   END_IF;
END_REGION

REGION Network 30: LBC_Axis64Pos Operation Mode
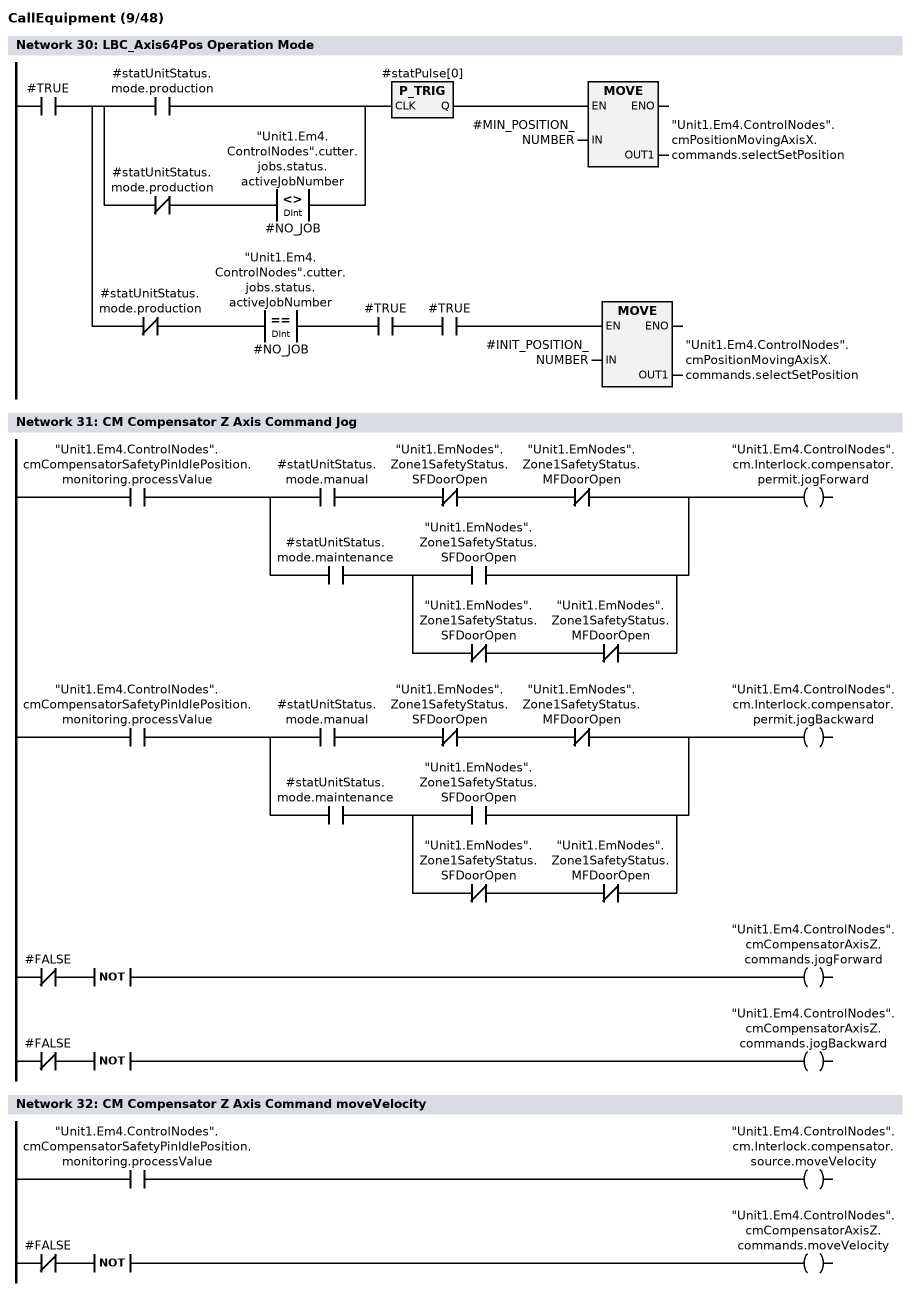
   RUNG wire#powerrail
      Contact( #TRUE )
      wire#w1
      Contact( #statUnitStatus.mode.production )
      wire#w2
      P_Trig( #statPulse[0] )
      Move(in := #MIN_POSITION_NUMBER, out1 => "Unit1.Em4.ControlNodes".cmPositionMovingAxisX.commands.selectSetPosition)
   END_RUNG
   RUNG wire#w1
      I_Contact( #statUnitStatus.mode.production )
      { S7_Templates := "SrcType := DInt" } NE_Contact(in1 := "Unit1.Em4.ControlNodes".cutter.jobs.status.activeJobNumber, in2 := #NO_JOB)
   END_RUNG wire#w2
   RUNG wire#w1
      I_Contact( #statUnitStatus.mode.production )
      { S7_Templates := "SrcType := DInt" } EQ_Contact(in1 := "Unit1.Em4.ControlNodes".cutter.jobs.status.activeJobNumber, in2 := #NO_JOB)
      Contact( #TRUE )
      Contact( #TRUE )
      Move(in := #INIT_POSITION_NUMBER, out1 => "Unit1.Em4.ControlNodes".cmPositionMovingAxisX.commands.selectSetPosition)
   END_RUNG
   // the same network as SCL:
   #_w1 := #TRUE AND (#statUnitStatus.mode.production OR (NOT #statUnitStatus.mode.production AND ("Unit1.Em4.ControlNodes".cutter.jobs.status.activeJobNumber <> #NO_JOB)));
   #_w2 := #_w1 AND NOT #statPulse[0];   // rising edge
   #statPulse[0] := #_w1;
   IF #_w2 THEN
       "Unit1.Em4.ControlNodes".cmPositionMovingAxisX.commands.selectSetPosition := #MIN_POSITION_NUMBER;
   END_IF;
   IF #TRUE AND NOT #statUnitStatus.mode.production AND ("Unit1.Em4.ControlNodes".cutter.jobs.status.activeJobNumber = #NO_JOB) AND #TRUE AND #TRUE THEN
       "Unit1.Em4.ControlNodes".cmPositionMovingAxisX.commands.selectSetPosition := #INIT_POSITION_NUMBER;
   END_IF;
END_REGION

REGION Network 31: CM Compensator Z Axis Command Jog
   RUNG wire#powerrail
      Contact( "Unit1.Em4.ControlNodes".cmCompensatorSafetyPinIdlePosition.monitoring.processValue )
      wire#w1
      Contact( #statUnitStatus.mode.manual )
      I_Contact( "Unit1.EmNodes".Zone1SafetyStatus.SFDoorOpen )
      I_Contact( "Unit1.EmNodes".Zone1SafetyStatus.MFDoorOpen )
      wire#w2
      Coil( "Unit1.Em4.ControlNodes".cm.Interlock.compensator.permit.jogForward )
   END_RUNG
   RUNG wire#w1
      Contact( #statUnitStatus.mode.maintenance )
      wire#w3
      Contact( "Unit1.EmNodes".Zone1SafetyStatus.SFDoorOpen )
   END_RUNG wire#w2
   RUNG wire#w3
      I_Contact( "Unit1.EmNodes".Zone1SafetyStatus.SFDoorOpen )
      I_Contact( "Unit1.EmNodes".Zone1SafetyStatus.MFDoorOpen )
   END_RUNG wire#w2
   RUNG wire#powerrail
      Contact( "Unit1.Em4.ControlNodes".cmCompensatorSafetyPinIdlePosition.monitoring.processValue )
      wire#w4
      Contact( #statUnitStatus.mode.manual )
      I_Contact( "Unit1.EmNodes".Zone1SafetyStatus.SFDoorOpen )
      I_Contact( "Unit1.EmNodes".Zone1SafetyStatus.MFDoorOpen )
      wire#w5
      Coil( "Unit1.Em4.ControlNodes".cm.Interlock.compensator.permit.jogBackward )
   END_RUNG
   RUNG wire#w4
      Contact( #statUnitStatus.mode.maintenance )
      wire#w6
      Contact( "Unit1.EmNodes".Zone1SafetyStatus.SFDoorOpen )
   END_RUNG wire#w5
   RUNG wire#w6
      I_Contact( "Unit1.EmNodes".Zone1SafetyStatus.SFDoorOpen )
      I_Contact( "Unit1.EmNodes".Zone1SafetyStatus.MFDoorOpen )
   END_RUNG wire#w5
   RUNG wire#powerrail
      I_Contact( #FALSE )
      Not()
      Coil( "Unit1.Em4.ControlNodes".cmCompensatorAxisZ.commands.jogForward )
   END_RUNG
   RUNG wire#powerrail
      I_Contact( #FALSE )
      Not()
      Coil( "Unit1.Em4.ControlNodes".cmCompensatorAxisZ.commands.jogBackward )
   END_RUNG
   // the same network as SCL:
   "Unit1.Em4.ControlNodes".cm.Interlock.compensator.permit.jogForward := "Unit1.Em4.ControlNodes".cmCompensatorSafetyPinIdlePosition.monitoring.processValue AND ((#statUnitStatus.mode.manual AND NOT "Unit1.EmNodes".Zone1SafetyStatus.SFDoorOpen AND NOT "Unit1.EmNodes".Zone1SafetyStatus.MFDoorOpen) OR (#statUnitStatus.mode.maintenance AND ("Unit1.EmNodes".Zone1SafetyStatus.SFDoorOpen OR (NOT "Unit1.EmNodes".Zone1SafetyStatus.SFDoorOpen AND NOT "Unit1.EmNodes".Zone1SafetyStatus.MFDoorOpen))));
   "Unit1.Em4.ControlNodes".cm.Interlock.compensator.permit.jogBackward := "Unit1.Em4.ControlNodes".cmCompensatorSafetyPinIdlePosition.monitoring.processValue AND ((#statUnitStatus.mode.manual AND NOT "Unit1.EmNodes".Zone1SafetyStatus.SFDoorOpen AND NOT "Unit1.EmNodes".Zone1SafetyStatus.MFDoorOpen) OR (#statUnitStatus.mode.maintenance AND ("Unit1.EmNodes".Zone1SafetyStatus.SFDoorOpen OR (NOT "Unit1.EmNodes".Zone1SafetyStatus.SFDoorOpen AND NOT "Unit1.EmNodes".Zone1SafetyStatus.MFDoorOpen))));
   "Unit1.Em4.ControlNodes".cmCompensatorAxisZ.commands.jogForward := NOT (NOT #FALSE);
   "Unit1.Em4.ControlNodes".cmCompensatorAxisZ.commands.jogBackward := NOT (NOT #FALSE);
END_REGION

REGION Network 32: CM Compensator Z Axis Command moveVelocity
   RUNG wire#powerrail
      Contact( "Unit1.Em4.ControlNodes".cmCompensatorSafetyPinIdlePosition.monitoring.processValue )
      Coil( "Unit1.Em4.ControlNodes".cm.Interlock.compensator.source.moveVelocity )
   END_RUNG
   RUNG wire#powerrail
      I_Contact( #FALSE )
      Not()
      Coil( "Unit1.Em4.ControlNodes".cmCompensatorAxisZ.commands.moveVelocity )
   END_RUNG
   // the same network as SCL:
   "Unit1.Em4.ControlNodes".cm.Interlock.compensator.source.moveVelocity := "Unit1.Em4.ControlNodes".cmCompensatorSafetyPinIdlePosition.monitoring.processValue;
   "Unit1.Em4.ControlNodes".cmCompensatorAxisZ.commands.moveVelocity := NOT (NOT #FALSE);
END_REGION

REGION Network 33: CM Compensator Z Axis Command stop
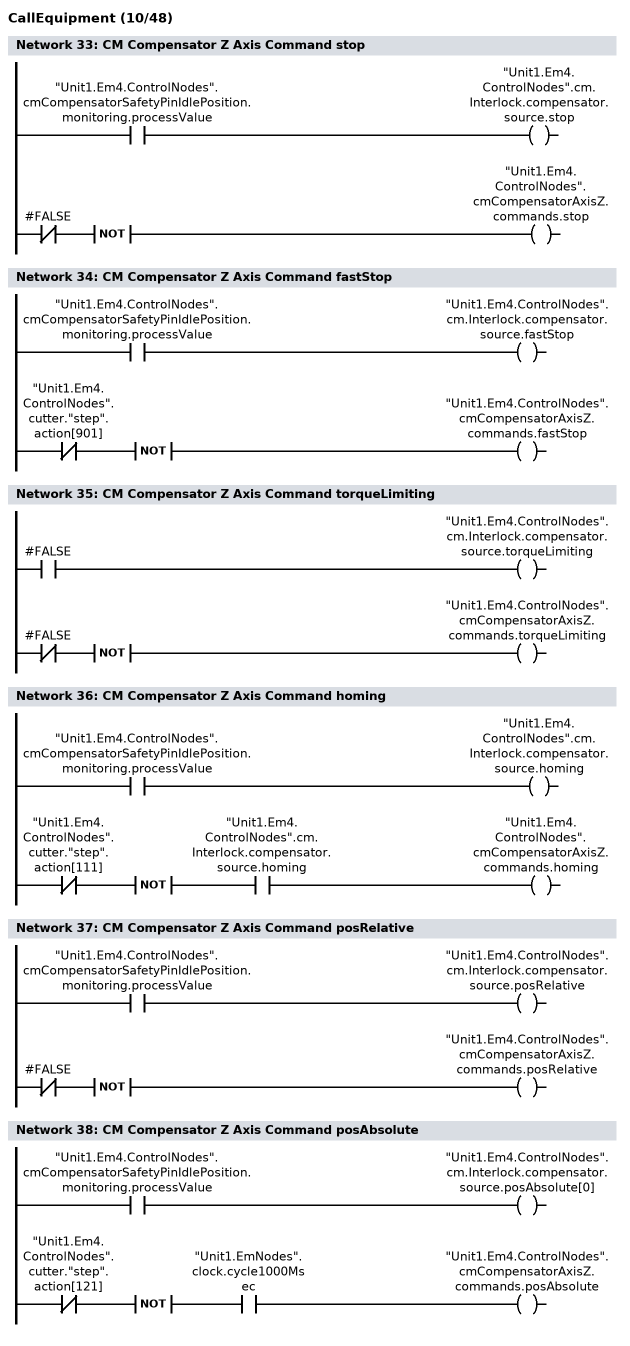
   RUNG wire#powerrail
      Contact( "Unit1.Em4.ControlNodes".cmCompensatorSafetyPinIdlePosition.monitoring.processValue )
      Coil( "Unit1.Em4.ControlNodes".cm.Interlock.compensator.source.stop )
   END_RUNG
   RUNG wire#powerrail
      I_Contact( #FALSE )
      Not()
      Coil( "Unit1.Em4.ControlNodes".cmCompensatorAxisZ.commands.stop )
   END_RUNG
   // the same network as SCL:
   "Unit1.Em4.ControlNodes".cm.Interlock.compensator.source.stop := "Unit1.Em4.ControlNodes".cmCompensatorSafetyPinIdlePosition.monitoring.processValue;
   "Unit1.Em4.ControlNodes".cmCompensatorAxisZ.commands.stop := NOT (NOT #FALSE);
END_REGION

REGION Network 34: CM Compensator Z Axis Command fastStop
   RUNG wire#powerrail
      Contact( "Unit1.Em4.ControlNodes".cmCompensatorSafetyPinIdlePosition.monitoring.processValue )
      Coil( "Unit1.Em4.ControlNodes".cm.Interlock.compensator.source.fastStop )
   END_RUNG
   RUNG wire#powerrail
      I_Contact( "Unit1.Em4.ControlNodes".cutter."step".action[901] )
      Not()
      Coil( "Unit1.Em4.ControlNodes".cmCompensatorAxisZ.commands.fastStop )
   END_RUNG
   // the same network as SCL:
   "Unit1.Em4.ControlNodes".cm.Interlock.compensator.source.fastStop := "Unit1.Em4.ControlNodes".cmCompensatorSafetyPinIdlePosition.monitoring.processValue;
   "Unit1.Em4.ControlNodes".cmCompensatorAxisZ.commands.fastStop := NOT (NOT "Unit1.Em4.ControlNodes".cutter."step".action[901]);
END_REGION

REGION Network 35: CM Compensator Z Axis Command torqueLimiting
   RUNG wire#powerrail
      Contact( #FALSE )
      Coil( "Unit1.Em4.ControlNodes".cm.Interlock.compensator.source.torqueLimiting )
   END_RUNG
   RUNG wire#powerrail
      I_Contact( #FALSE )
      Not()
      Coil( "Unit1.Em4.ControlNodes".cmCompensatorAxisZ.commands.torqueLimiting )
   END_RUNG
   // the same network as SCL:
   "Unit1.Em4.ControlNodes".cm.Interlock.compensator.source.torqueLimiting := #FALSE;
   "Unit1.Em4.ControlNodes".cmCompensatorAxisZ.commands.torqueLimiting := NOT (NOT #FALSE);
END_REGION

REGION Network 36: CM Compensator Z Axis Command homing
   RUNG wire#powerrail
      Contact( "Unit1.Em4.ControlNodes".cmCompensatorSafetyPinIdlePosition.monitoring.processValue )
      Coil( "Unit1.Em4.ControlNodes".cm.Interlock.compensator.source.homing )
   END_RUNG
   RUNG wire#powerrail
      I_Contact( "Unit1.Em4.ControlNodes".cutter."step".action[111] )
      Not()
      Contact( "Unit1.Em4.ControlNodes".cm.Interlock.compensator.source.homing )
      Coil( "Unit1.Em4.ControlNodes".cmCompensatorAxisZ.commands.homing )
   END_RUNG
   // the same network as SCL:
   "Unit1.Em4.ControlNodes".cm.Interlock.compensator.source.homing := "Unit1.Em4.ControlNodes".cmCompensatorSafetyPinIdlePosition.monitoring.processValue;
   "Unit1.Em4.ControlNodes".cmCompensatorAxisZ.commands.homing := NOT (NOT "Unit1.Em4.ControlNodes".cutter."step".action[111]) AND "Unit1.Em4.ControlNodes".cm.Interlock.compensator.source.homing;
END_REGION

REGION Network 37: CM Compensator Z Axis Command posRelative
   RUNG wire#powerrail
      Contact( "Unit1.Em4.ControlNodes".cmCompensatorSafetyPinIdlePosition.monitoring.processValue )
      Coil( "Unit1.Em4.ControlNodes".cm.Interlock.compensator.source.posRelative )
   END_RUNG
   RUNG wire#powerrail
      I_Contact( #FALSE )
      Not()
      Coil( "Unit1.Em4.ControlNodes".cmCompensatorAxisZ.commands.posRelative )
   END_RUNG
   // the same network as SCL:
   "Unit1.Em4.ControlNodes".cm.Interlock.compensator.source.posRelative := "Unit1.Em4.ControlNodes".cmCompensatorSafetyPinIdlePosition.monitoring.processValue;
   "Unit1.Em4.ControlNodes".cmCompensatorAxisZ.commands.posRelative := NOT (NOT #FALSE);
END_REGION

REGION Network 38: CM Compensator Z Axis Command posAbsolute
   RUNG wire#powerrail
      Contact( "Unit1.Em4.ControlNodes".cmCompensatorSafetyPinIdlePosition.monitoring.processValue )
      Coil( "Unit1.Em4.ControlNodes".cm.Interlock.compensator.source.posAbsolute[0] )
   END_RUNG
   RUNG wire#powerrail
      I_Contact( "Unit1.Em4.ControlNodes".cutter."step".action[121] )
      Not()
      Contact( "Unit1.EmNodes".clock.cycle1000Msec )
      Coil( "Unit1.Em4.ControlNodes".cmCompensatorAxisZ.commands.posAbsolute )
   END_RUNG
   // the same network as SCL:
   "Unit1.Em4.ControlNodes".cm.Interlock.compensator.source.posAbsolute[0] := "Unit1.Em4.ControlNodes".cmCompensatorSafetyPinIdlePosition.monitoring.processValue;
   "Unit1.Em4.ControlNodes".cmCompensatorAxisZ.commands.posAbsolute := NOT (NOT "Unit1.Em4.ControlNodes".cutter."step".action[121]) AND "Unit1.EmNodes".clock.cycle1000Msec;
END_REGION

REGION Network 39: CM Compensator Z Axis Command gearInRelative
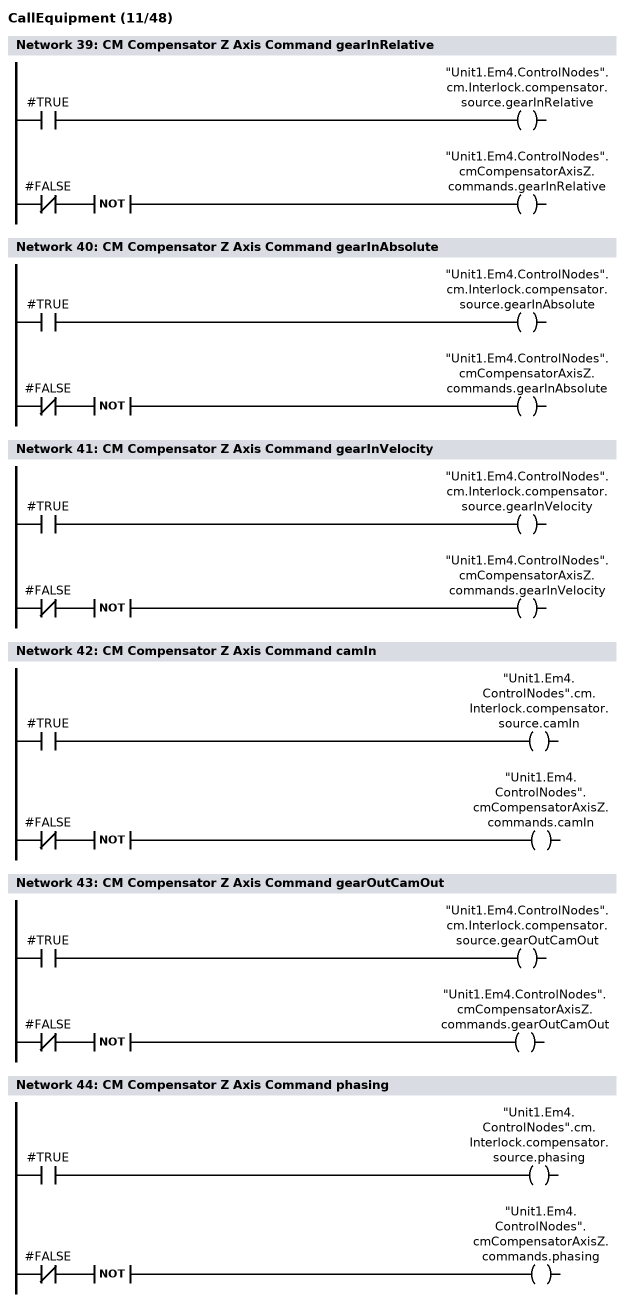
   RUNG wire#powerrail
      Contact( #TRUE )
      Coil( "Unit1.Em4.ControlNodes".cm.Interlock.compensator.source.gearInRelative )
   END_RUNG
   RUNG wire#powerrail
      I_Contact( #FALSE )
      Not()
      Coil( "Unit1.Em4.ControlNodes".cmCompensatorAxisZ.commands.gearInRelative )
   END_RUNG
   // the same network as SCL:
   "Unit1.Em4.ControlNodes".cm.Interlock.compensator.source.gearInRelative := #TRUE;
   "Unit1.Em4.ControlNodes".cmCompensatorAxisZ.commands.gearInRelative := NOT (NOT #FALSE);
END_REGION

REGION Network 40: CM Compensator Z Axis Command gearInAbsolute
   RUNG wire#powerrail
      Contact( #TRUE )
      Coil( "Unit1.Em4.ControlNodes".cm.Interlock.compensator.source.gearInAbsolute )
   END_RUNG
   RUNG wire#powerrail
      I_Contact( #FALSE )
      Not()
      Coil( "Unit1.Em4.ControlNodes".cmCompensatorAxisZ.commands.gearInAbsolute )
   END_RUNG
   // the same network as SCL:
   "Unit1.Em4.ControlNodes".cm.Interlock.compensator.source.gearInAbsolute := #TRUE;
   "Unit1.Em4.ControlNodes".cmCompensatorAxisZ.commands.gearInAbsolute := NOT (NOT #FALSE);
END_REGION

REGION Network 41: CM Compensator Z Axis Command gearInVelocity
   RUNG wire#powerrail
      Contact( #TRUE )
      Coil( "Unit1.Em4.ControlNodes".cm.Interlock.compensator.source.gearInVelocity )
   END_RUNG
   RUNG wire#powerrail
      I_Contact( #FALSE )
      Not()
      Coil( "Unit1.Em4.ControlNodes".cmCompensatorAxisZ.commands.gearInVelocity )
   END_RUNG
   // the same network as SCL:
   "Unit1.Em4.ControlNodes".cm.Interlock.compensator.source.gearInVelocity := #TRUE;
   "Unit1.Em4.ControlNodes".cmCompensatorAxisZ.commands.gearInVelocity := NOT (NOT #FALSE);
END_REGION

REGION Network 42: CM Compensator Z Axis Command camIn
   RUNG wire#powerrail
      Contact( #TRUE )
      Coil( "Unit1.Em4.ControlNodes".cm.Interlock.compensator.source.camIn )
   END_RUNG
   RUNG wire#powerrail
      I_Contact( #FALSE )
      Not()
      Coil( "Unit1.Em4.ControlNodes".cmCompensatorAxisZ.commands.camIn )
   END_RUNG
   // the same network as SCL:
   "Unit1.Em4.ControlNodes".cm.Interlock.compensator.source.camIn := #TRUE;
   "Unit1.Em4.ControlNodes".cmCompensatorAxisZ.commands.camIn := NOT (NOT #FALSE);
END_REGION

REGION Network 43: CM Compensator Z Axis Command gearOutCamOut
   RUNG wire#powerrail
      Contact( #TRUE )
      Coil( "Unit1.Em4.ControlNodes".cm.Interlock.compensator.source.gearOutCamOut )
   END_RUNG
   RUNG wire#powerrail
      I_Contact( #FALSE )
      Not()
      Coil( "Unit1.Em4.ControlNodes".cmCompensatorAxisZ.commands.gearOutCamOut )
   END_RUNG
   // the same network as SCL:
   "Unit1.Em4.ControlNodes".cm.Interlock.compensator.source.gearOutCamOut := #TRUE;
   "Unit1.Em4.ControlNodes".cmCompensatorAxisZ.commands.gearOutCamOut := NOT (NOT #FALSE);
END_REGION

REGION Network 44: CM Compensator Z Axis Command phasing
   RUNG wire#powerrail
      Contact( #TRUE )
      Coil( "Unit1.Em4.ControlNodes".cm.Interlock.compensator.source.phasing )
   END_RUNG
   RUNG wire#powerrail
      I_Contact( #FALSE )
      Not()
      Coil( "Unit1.Em4.ControlNodes".cmCompensatorAxisZ.commands.phasing )
   END_RUNG
   // the same network as SCL:
   "Unit1.Em4.ControlNodes".cm.Interlock.compensator.source.phasing := #TRUE;
   "Unit1.Em4.ControlNodes".cmCompensatorAxisZ.commands.phasing := NOT (NOT #FALSE);
END_REGION

REGION Network 45: CM Compensator Z Axis Command offset
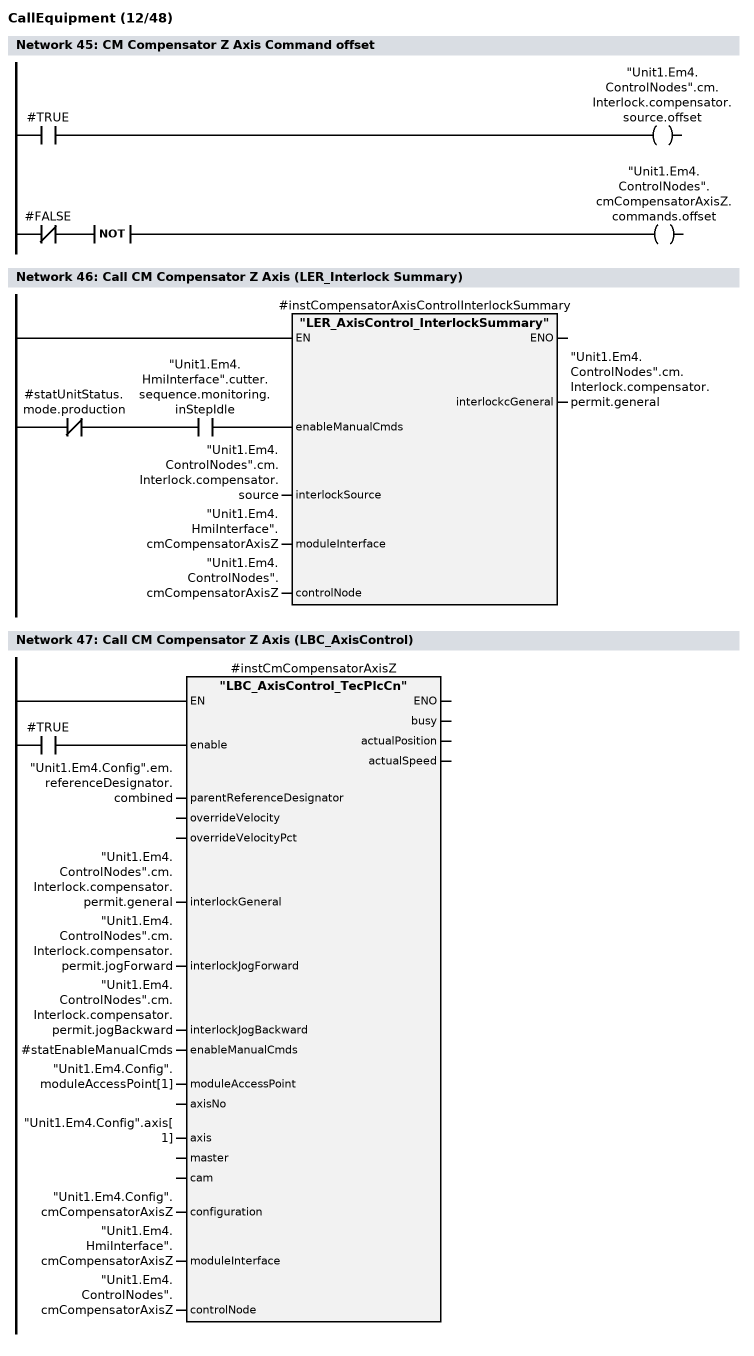
   RUNG wire#powerrail
      Contact( #TRUE )
      Coil( "Unit1.Em4.ControlNodes".cm.Interlock.compensator.source.offset )
   END_RUNG
   RUNG wire#powerrail
      I_Contact( #FALSE )
      Not()
      Coil( "Unit1.Em4.ControlNodes".cmCompensatorAxisZ.commands.offset )
   END_RUNG
   // the same network as SCL:
   "Unit1.Em4.ControlNodes".cm.Interlock.compensator.source.offset := #TRUE;
   "Unit1.Em4.ControlNodes".cmCompensatorAxisZ.commands.offset := NOT (NOT #FALSE);
END_REGION

REGION Network 46: Call CM Compensator Z Axis (LER_Interlock Summary)
   RUNG wire#powerrail
      #instCompensatorAxisControlInterlockSummary(enableManualCmds := wire#w1, interlockSource := "Unit1.Em4.ControlNodes".cm.Interlock.compensator.source, moduleInterface := "Unit1.Em4.HmiInterface".cmCompensatorAxisZ, controlNode := "Unit1.Em4.ControlNodes".cmCompensatorAxisZ, interlockcGeneral => "Unit1.Em4.ControlNodes".cm.Interlock.compensator.permit.general)
   END_RUNG
   RUNG wire#powerrail
      I_Contact( #statUnitStatus.mode.production )
      Contact( "Unit1.Em4.HmiInterface".cutter.sequence.monitoring.inStepIdle )
   END_RUNG wire#w1
   // the same network as SCL:
   #instCompensatorAxisControlInterlockSummary(enableManualCmds := NOT #statUnitStatus.mode.production AND "Unit1.Em4.HmiInterface".cutter.sequence.monitoring.inStepIdle,   // "LER_AxisControl_InterlockSummary"
                           interlockSource := "Unit1.Em4.ControlNodes".cm.Interlock.compensator.source,
                           moduleInterface := "Unit1.Em4.HmiInterface".cmCompensatorAxisZ,
                           controlNode := "Unit1.Em4.ControlNodes".cmCompensatorAxisZ,
                           interlockcGeneral => "Unit1.Em4.ControlNodes".cm.Interlock.compensator.permit.general);
END_REGION

REGION Network 47: Call CM Compensator Z Axis (LBC_AxisControl)
   RUNG wire#powerrail
      #instCmCompensatorAxisZ(enable := wire#w1, parentReferenceDesignator := "Unit1.Em4.Config".em.referenceDesignator.combined, overrideVelocity :=, overrideVelocityPct :=, interlockGeneral := "Unit1.Em4.ControlNodes".cm.Interlock.compensator.permit.general, interlockJogForward := "Unit1.Em4.ControlNodes".cm.Interlock.compensator.permit.jogForward, interlockJogBackward := "Unit1.Em4.ControlNodes".cm.Interlock.compensator.permit.jogBackward, enableManualCmds := #statEnableManualCmds, moduleAccessPoint := "Unit1.Em4.Config".moduleAccessPoint[1], axisNo :=, axis := "Unit1.Em4.Config".axis[1], master :=, cam :=, configuration := "Unit1.Em4.Config".cmCompensatorAxisZ, moduleInterface := "Unit1.Em4.HmiInterface".cmCompensatorAxisZ, controlNode := "Unit1.Em4.ControlNodes".cmCompensatorAxisZ, busy =>, actualPosition =>, actualSpeed =>)
   END_RUNG
   RUNG wire#powerrail
      Contact( #TRUE )
   END_RUNG wire#w1
   // the same network as SCL:
   #instCmCompensatorAxisZ(enable := #TRUE,   // "LBC_AxisControl_TecPlcCn"
                           parentReferenceDesignator := "Unit1.Em4.Config".em.referenceDesignator.combined,
                           interlockGeneral := "Unit1.Em4.ControlNodes".cm.Interlock.compensator.permit.general,
                           interlockJogForward := "Unit1.Em4.ControlNodes".cm.Interlock.compensator.permit.jogForward,
                           interlockJogBackward := "Unit1.Em4.ControlNodes".cm.Interlock.compensator.permit.jogBackward,
                           enableManualCmds := #statEnableManualCmds,
                           moduleAccessPoint := "Unit1.Em4.Config".moduleAccessPoint[1],
                           axis := "Unit1.Em4.Config".axis[1],
                           configuration := "Unit1.Em4.Config".cmCompensatorAxisZ,
                           moduleInterface := "Unit1.Em4.HmiInterface".cmCompensatorAxisZ,
                           controlNode := "Unit1.Em4.ControlNodes".cmCompensatorAxisZ);
END_REGION

REGION Network 48: Call CM Compensator Z Axis (LER_ServoTorqueCal)
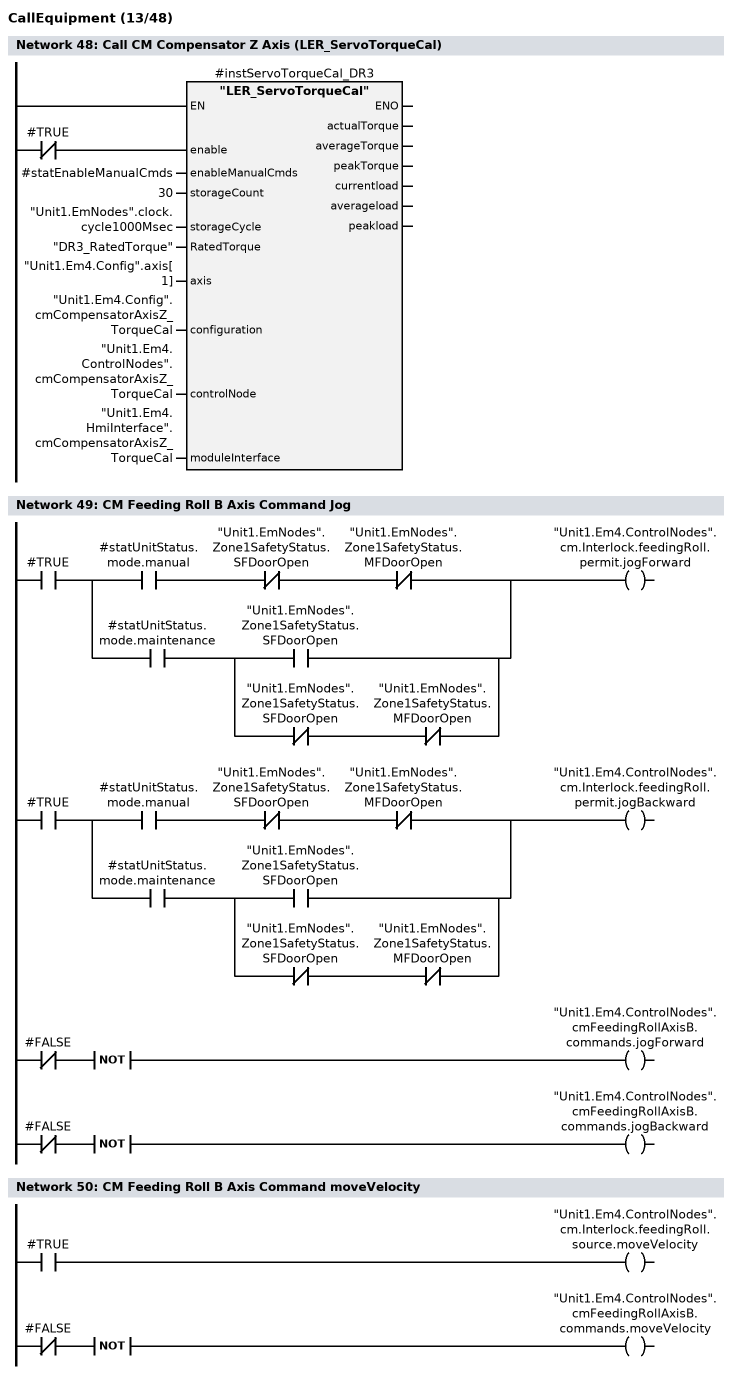
   RUNG wire#powerrail
      #instServoTorqueCal_DR3(enable := wire#w1, enableManualCmds := #statEnableManualCmds, storageCount := 30, storageCycle := "Unit1.EmNodes".clock.cycle1000Msec, RatedTorque := "DR3_RatedTorque", axis := "Unit1.Em4.Config".axis[1], configuration := "Unit1.Em4.Config".cmCompensatorAxisZ_TorqueCal, controlNode := "Unit1.Em4.ControlNodes".cmCompensatorAxisZ_TorqueCal, moduleInterface := "Unit1.Em4.HmiInterface".cmCompensatorAxisZ_TorqueCal, actualTorque =>, averageTorque =>, peakTorque =>, currentload =>, averageload =>, peakload =>)
   END_RUNG
   RUNG wire#powerrail
      I_Contact( #TRUE )
   END_RUNG wire#w1
   // the same network as SCL:
   #instServoTorqueCal_DR3(enable := NOT #TRUE,   // "LER_ServoTorqueCal"
                           enableManualCmds := #statEnableManualCmds,
                           storageCount := 30,
                           storageCycle := "Unit1.EmNodes".clock.cycle1000Msec,
                           RatedTorque := "DR3_RatedTorque",
                           axis := "Unit1.Em4.Config".axis[1],
                           configuration := "Unit1.Em4.Config".cmCompensatorAxisZ_TorqueCal,
                           controlNode := "Unit1.Em4.ControlNodes".cmCompensatorAxisZ_TorqueCal,
                           moduleInterface := "Unit1.Em4.HmiInterface".cmCompensatorAxisZ_TorqueCal);
END_REGION

REGION Network 49: CM Feeding Roll B Axis Command Jog
   RUNG wire#powerrail
      Contact( #TRUE )
      wire#w1
      Contact( #statUnitStatus.mode.manual )
      I_Contact( "Unit1.EmNodes".Zone1SafetyStatus.SFDoorOpen )
      I_Contact( "Unit1.EmNodes".Zone1SafetyStatus.MFDoorOpen )
      wire#w2
      Coil( "Unit1.Em4.ControlNodes".cm.Interlock.feedingRoll.permit.jogForward )
   END_RUNG
   RUNG wire#w1
      Contact( #statUnitStatus.mode.maintenance )
      wire#w3
      Contact( "Unit1.EmNodes".Zone1SafetyStatus.SFDoorOpen )
   END_RUNG wire#w2
   RUNG wire#w3
      I_Contact( "Unit1.EmNodes".Zone1SafetyStatus.SFDoorOpen )
      I_Contact( "Unit1.EmNodes".Zone1SafetyStatus.MFDoorOpen )
   END_RUNG wire#w2
   RUNG wire#powerrail
      Contact( #TRUE )
      wire#w4
      Contact( #statUnitStatus.mode.manual )
      I_Contact( "Unit1.EmNodes".Zone1SafetyStatus.SFDoorOpen )
      I_Contact( "Unit1.EmNodes".Zone1SafetyStatus.MFDoorOpen )
      wire#w5
      Coil( "Unit1.Em4.ControlNodes".cm.Interlock.feedingRoll.permit.jogBackward )
   END_RUNG
   RUNG wire#w4
      Contact( #statUnitStatus.mode.maintenance )
      wire#w6
      Contact( "Unit1.EmNodes".Zone1SafetyStatus.SFDoorOpen )
   END_RUNG wire#w5
   RUNG wire#w6
      I_Contact( "Unit1.EmNodes".Zone1SafetyStatus.SFDoorOpen )
      I_Contact( "Unit1.EmNodes".Zone1SafetyStatus.MFDoorOpen )
   END_RUNG wire#w5
   RUNG wire#powerrail
      I_Contact( #FALSE )
      Not()
      Coil( "Unit1.Em4.ControlNodes".cmFeedingRollAxisB.commands.jogForward )
   END_RUNG
   RUNG wire#powerrail
      I_Contact( #FALSE )
      Not()
      Coil( "Unit1.Em4.ControlNodes".cmFeedingRollAxisB.commands.jogBackward )
   END_RUNG
   // the same network as SCL:
   "Unit1.Em4.ControlNodes".cm.Interlock.feedingRoll.permit.jogForward := #TRUE AND ((#statUnitStatus.mode.manual AND NOT "Unit1.EmNodes".Zone1SafetyStatus.SFDoorOpen AND NOT "Unit1.EmNodes".Zone1SafetyStatus.MFDoorOpen) OR (#statUnitStatus.mode.maintenance AND ("Unit1.EmNodes".Zone1SafetyStatus.SFDoorOpen OR (NOT "Unit1.EmNodes".Zone1SafetyStatus.SFDoorOpen AND NOT "Unit1.EmNodes".Zone1SafetyStatus.MFDoorOpen))));
   "Unit1.Em4.ControlNodes".cm.Interlock.feedingRoll.permit.jogBackward := #TRUE AND ((#statUnitStatus.mode.manual AND NOT "Unit1.EmNodes".Zone1SafetyStatus.SFDoorOpen AND NOT "Unit1.EmNodes".Zone1SafetyStatus.MFDoorOpen) OR (#statUnitStatus.mode.maintenance AND ("Unit1.EmNodes".Zone1SafetyStatus.SFDoorOpen OR (NOT "Unit1.EmNodes".Zone1SafetyStatus.SFDoorOpen AND NOT "Unit1.EmNodes".Zone1SafetyStatus.MFDoorOpen))));
   "Unit1.Em4.ControlNodes".cmFeedingRollAxisB.commands.jogForward := NOT (NOT #FALSE);
   "Unit1.Em4.ControlNodes".cmFeedingRollAxisB.commands.jogBackward := NOT (NOT #FALSE);
END_REGION

REGION Network 50: CM Feeding Roll B Axis Command moveVelocity
   RUNG wire#powerrail
      Contact( #TRUE )
      Coil( "Unit1.Em4.ControlNodes".cm.Interlock.feedingRoll.source.moveVelocity )
   END_RUNG
   RUNG wire#powerrail
      I_Contact( #FALSE )
      Not()
      Coil( "Unit1.Em4.ControlNodes".cmFeedingRollAxisB.commands.moveVelocity )
   END_RUNG
   // the same network as SCL:
   "Unit1.Em4.ControlNodes".cm.Interlock.feedingRoll.source.moveVelocity := #TRUE;
   "Unit1.Em4.ControlNodes".cmFeedingRollAxisB.commands.moveVelocity := NOT (NOT #FALSE);
END_REGION

REGION Network 51: CM Feeding Roll B Axis Command stop
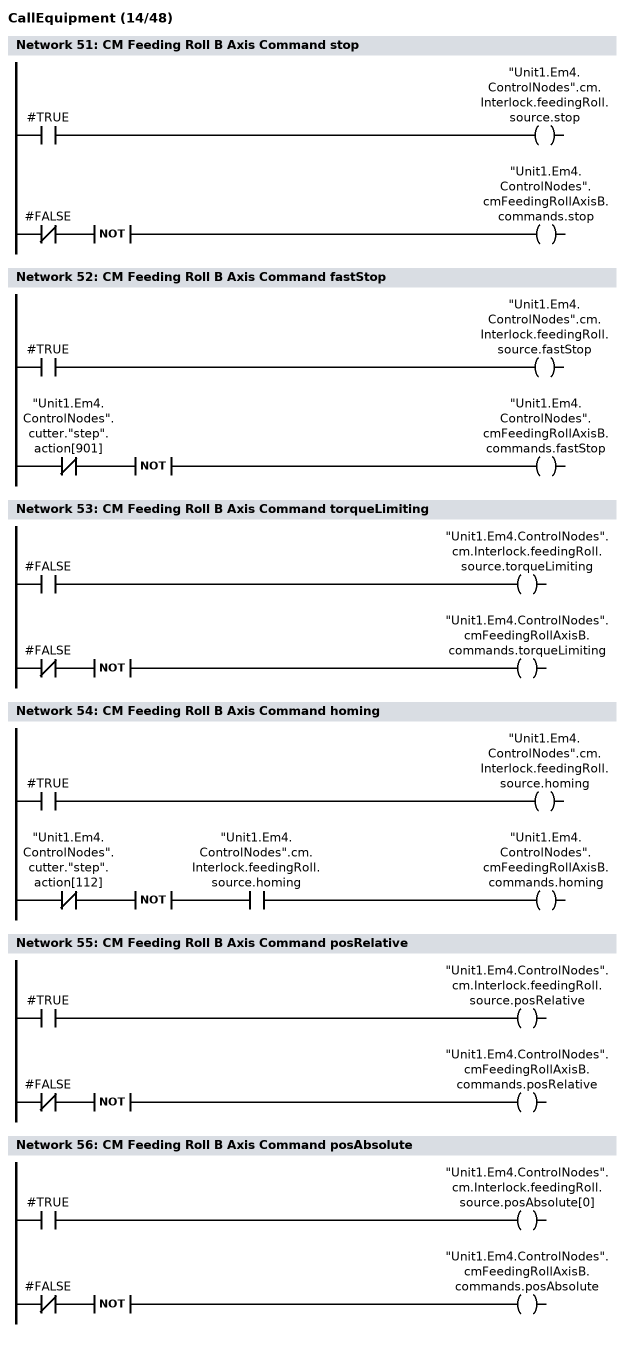
   RUNG wire#powerrail
      Contact( #TRUE )
      Coil( "Unit1.Em4.ControlNodes".cm.Interlock.feedingRoll.source.stop )
   END_RUNG
   RUNG wire#powerrail
      I_Contact( #FALSE )
      Not()
      Coil( "Unit1.Em4.ControlNodes".cmFeedingRollAxisB.commands.stop )
   END_RUNG
   // the same network as SCL:
   "Unit1.Em4.ControlNodes".cm.Interlock.feedingRoll.source.stop := #TRUE;
   "Unit1.Em4.ControlNodes".cmFeedingRollAxisB.commands.stop := NOT (NOT #FALSE);
END_REGION

REGION Network 52: CM Feeding Roll B Axis Command fastStop
   RUNG wire#powerrail
      Contact( #TRUE )
      Coil( "Unit1.Em4.ControlNodes".cm.Interlock.feedingRoll.source.fastStop )
   END_RUNG
   RUNG wire#powerrail
      I_Contact( "Unit1.Em4.ControlNodes".cutter."step".action[901] )
      Not()
      Coil( "Unit1.Em4.ControlNodes".cmFeedingRollAxisB.commands.fastStop )
   END_RUNG
   // the same network as SCL:
   "Unit1.Em4.ControlNodes".cm.Interlock.feedingRoll.source.fastStop := #TRUE;
   "Unit1.Em4.ControlNodes".cmFeedingRollAxisB.commands.fastStop := NOT (NOT "Unit1.Em4.ControlNodes".cutter."step".action[901]);
END_REGION

REGION Network 53: CM Feeding Roll B Axis Command torqueLimiting
   RUNG wire#powerrail
      Contact( #FALSE )
      Coil( "Unit1.Em4.ControlNodes".cm.Interlock.feedingRoll.source.torqueLimiting )
   END_RUNG
   RUNG wire#powerrail
      I_Contact( #FALSE )
      Not()
      Coil( "Unit1.Em4.ControlNodes".cmFeedingRollAxisB.commands.torqueLimiting )
   END_RUNG
   // the same network as SCL:
   "Unit1.Em4.ControlNodes".cm.Interlock.feedingRoll.source.torqueLimiting := #FALSE;
   "Unit1.Em4.ControlNodes".cmFeedingRollAxisB.commands.torqueLimiting := NOT (NOT #FALSE);
END_REGION

REGION Network 54: CM Feeding Roll B Axis Command homing
   RUNG wire#powerrail
      Contact( #TRUE )
      Coil( "Unit1.Em4.ControlNodes".cm.Interlock.feedingRoll.source.homing )
   END_RUNG
   RUNG wire#powerrail
      I_Contact( "Unit1.Em4.ControlNodes".cutter."step".action[112] )
      Not()
      Contact( "Unit1.Em4.ControlNodes".cm.Interlock.feedingRoll.source.homing )
      Coil( "Unit1.Em4.ControlNodes".cmFeedingRollAxisB.commands.homing )
   END_RUNG
   // the same network as SCL:
   "Unit1.Em4.ControlNodes".cm.Interlock.feedingRoll.source.homing := #TRUE;
   "Unit1.Em4.ControlNodes".cmFeedingRollAxisB.commands.homing := NOT (NOT "Unit1.Em4.ControlNodes".cutter."step".action[112]) AND "Unit1.Em4.ControlNodes".cm.Interlock.feedingRoll.source.homing;
END_REGION

REGION Network 55: CM Feeding Roll B Axis Command posRelative
   RUNG wire#powerrail
      Contact( #TRUE )
      Coil( "Unit1.Em4.ControlNodes".cm.Interlock.feedingRoll.source.posRelative )
   END_RUNG
   RUNG wire#powerrail
      I_Contact( #FALSE )
      Not()
      Coil( "Unit1.Em4.ControlNodes".cmFeedingRollAxisB.commands.posRelative )
   END_RUNG
   // the same network as SCL:
   "Unit1.Em4.ControlNodes".cm.Interlock.feedingRoll.source.posRelative := #TRUE;
   "Unit1.Em4.ControlNodes".cmFeedingRollAxisB.commands.posRelative := NOT (NOT #FALSE);
END_REGION

REGION Network 56: CM Feeding Roll B Axis Command posAbsolute
   RUNG wire#powerrail
      Contact( #TRUE )
      Coil( "Unit1.Em4.ControlNodes".cm.Interlock.feedingRoll.source.posAbsolute[0] )
   END_RUNG
   RUNG wire#powerrail
      I_Contact( #FALSE )
      Not()
      Coil( "Unit1.Em4.ControlNodes".cmFeedingRollAxisB.commands.posAbsolute )
   END_RUNG
   // the same network as SCL:
   "Unit1.Em4.ControlNodes".cm.Interlock.feedingRoll.source.posAbsolute[0] := #TRUE;
   "Unit1.Em4.ControlNodes".cmFeedingRollAxisB.commands.posAbsolute := NOT (NOT #FALSE);
END_REGION

REGION Network 57: CM Feeding Roll B Axis Command gearInRelative
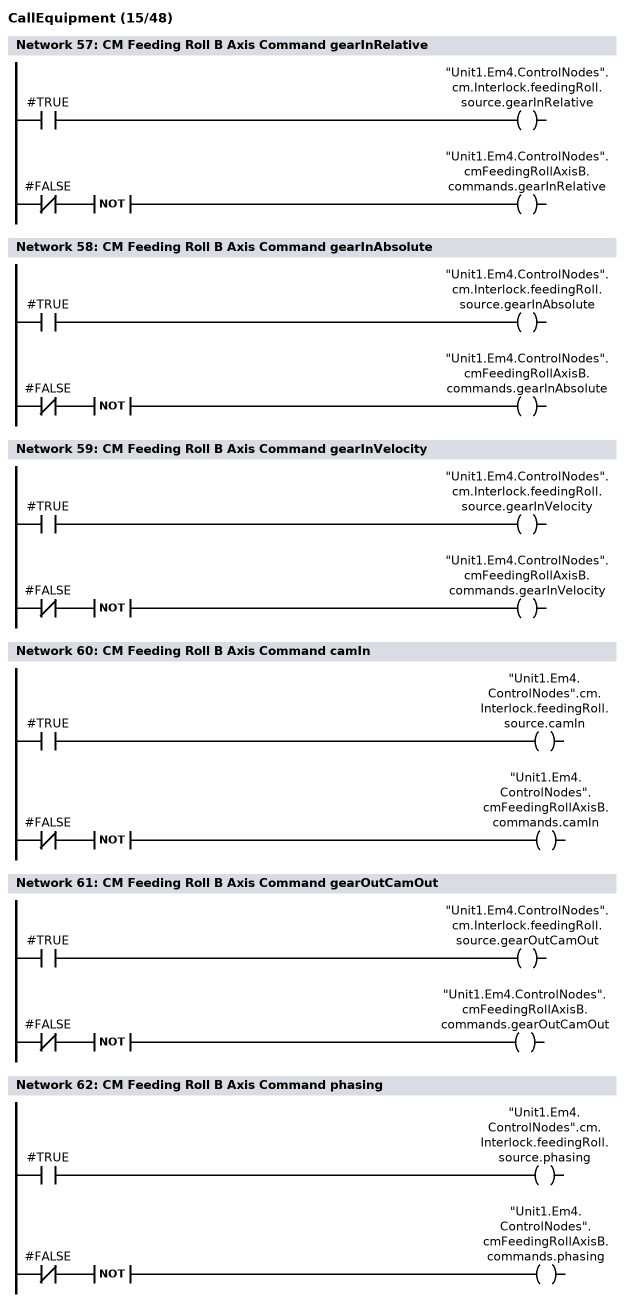
   RUNG wire#powerrail
      Contact( #TRUE )
      Coil( "Unit1.Em4.ControlNodes".cm.Interlock.feedingRoll.source.gearInRelative )
   END_RUNG
   RUNG wire#powerrail
      I_Contact( #FALSE )
      Not()
      Coil( "Unit1.Em4.ControlNodes".cmFeedingRollAxisB.commands.gearInRelative )
   END_RUNG
   // the same network as SCL:
   "Unit1.Em4.ControlNodes".cm.Interlock.feedingRoll.source.gearInRelative := #TRUE;
   "Unit1.Em4.ControlNodes".cmFeedingRollAxisB.commands.gearInRelative := NOT (NOT #FALSE);
END_REGION

REGION Network 58: CM Feeding Roll B Axis Command gearInAbsolute
   RUNG wire#powerrail
      Contact( #TRUE )
      Coil( "Unit1.Em4.ControlNodes".cm.Interlock.feedingRoll.source.gearInAbsolute )
   END_RUNG
   RUNG wire#powerrail
      I_Contact( #FALSE )
      Not()
      Coil( "Unit1.Em4.ControlNodes".cmFeedingRollAxisB.commands.gearInAbsolute )
   END_RUNG
   // the same network as SCL:
   "Unit1.Em4.ControlNodes".cm.Interlock.feedingRoll.source.gearInAbsolute := #TRUE;
   "Unit1.Em4.ControlNodes".cmFeedingRollAxisB.commands.gearInAbsolute := NOT (NOT #FALSE);
END_REGION

REGION Network 59: CM Feeding Roll B Axis Command gearInVelocity
   RUNG wire#powerrail
      Contact( #TRUE )
      Coil( "Unit1.Em4.ControlNodes".cm.Interlock.feedingRoll.source.gearInVelocity )
   END_RUNG
   RUNG wire#powerrail
      I_Contact( #FALSE )
      Not()
      Coil( "Unit1.Em4.ControlNodes".cmFeedingRollAxisB.commands.gearInVelocity )
   END_RUNG
   // the same network as SCL:
   "Unit1.Em4.ControlNodes".cm.Interlock.feedingRoll.source.gearInVelocity := #TRUE;
   "Unit1.Em4.ControlNodes".cmFeedingRollAxisB.commands.gearInVelocity := NOT (NOT #FALSE);
END_REGION

REGION Network 60: CM Feeding Roll B Axis Command camIn
   RUNG wire#powerrail
      Contact( #TRUE )
      Coil( "Unit1.Em4.ControlNodes".cm.Interlock.feedingRoll.source.camIn )
   END_RUNG
   RUNG wire#powerrail
      I_Contact( #FALSE )
      Not()
      Coil( "Unit1.Em4.ControlNodes".cmFeedingRollAxisB.commands.camIn )
   END_RUNG
   // the same network as SCL:
   "Unit1.Em4.ControlNodes".cm.Interlock.feedingRoll.source.camIn := #TRUE;
   "Unit1.Em4.ControlNodes".cmFeedingRollAxisB.commands.camIn := NOT (NOT #FALSE);
END_REGION

REGION Network 61: CM Feeding Roll B Axis Command gearOutCamOut
   RUNG wire#powerrail
      Contact( #TRUE )
      Coil( "Unit1.Em4.ControlNodes".cm.Interlock.feedingRoll.source.gearOutCamOut )
   END_RUNG
   RUNG wire#powerrail
      I_Contact( #FALSE )
      Not()
      Coil( "Unit1.Em4.ControlNodes".cmFeedingRollAxisB.commands.gearOutCamOut )
   END_RUNG
   // the same network as SCL:
   "Unit1.Em4.ControlNodes".cm.Interlock.feedingRoll.source.gearOutCamOut := #TRUE;
   "Unit1.Em4.ControlNodes".cmFeedingRollAxisB.commands.gearOutCamOut := NOT (NOT #FALSE);
END_REGION

REGION Network 62: CM Feeding Roll B Axis Command phasing
   RUNG wire#powerrail
      Contact( #TRUE )
      Coil( "Unit1.Em4.ControlNodes".cm.Interlock.feedingRoll.source.phasing )
   END_RUNG
   RUNG wire#powerrail
      I_Contact( #FALSE )
      Not()
      Coil( "Unit1.Em4.ControlNodes".cmFeedingRollAxisB.commands.phasing )
   END_RUNG
   // the same network as SCL:
   "Unit1.Em4.ControlNodes".cm.Interlock.feedingRoll.source.phasing := #TRUE;
   "Unit1.Em4.ControlNodes".cmFeedingRollAxisB.commands.phasing := NOT (NOT #FALSE);
END_REGION

REGION Network 63: CM Feeding Roll B Axis Command offset
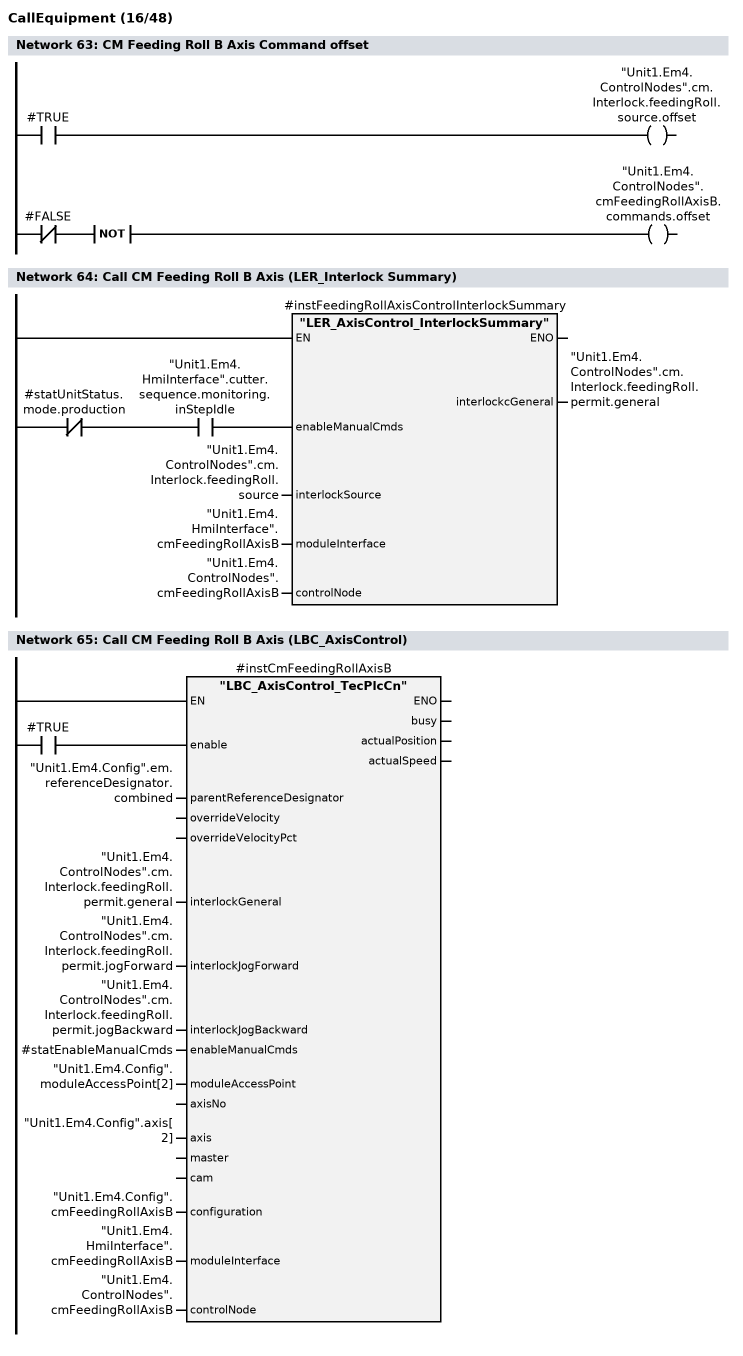
   RUNG wire#powerrail
      Contact( #TRUE )
      Coil( "Unit1.Em4.ControlNodes".cm.Interlock.feedingRoll.source.offset )
   END_RUNG
   RUNG wire#powerrail
      I_Contact( #FALSE )
      Not()
      Coil( "Unit1.Em4.ControlNodes".cmFeedingRollAxisB.commands.offset )
   END_RUNG
   // the same network as SCL:
   "Unit1.Em4.ControlNodes".cm.Interlock.feedingRoll.source.offset := #TRUE;
   "Unit1.Em4.ControlNodes".cmFeedingRollAxisB.commands.offset := NOT (NOT #FALSE);
END_REGION

REGION Network 64: Call CM Feeding Roll B Axis (LER_Interlock Summary)
   RUNG wire#powerrail
      #instFeedingRollAxisControlInterlockSummary(enableManualCmds := wire#w1, interlockSource := "Unit1.Em4.ControlNodes".cm.Interlock.feedingRoll.source, moduleInterface := "Unit1.Em4.HmiInterface".cmFeedingRollAxisB, controlNode := "Unit1.Em4.ControlNodes".cmFeedingRollAxisB, interlockcGeneral => "Unit1.Em4.ControlNodes".cm.Interlock.feedingRoll.permit.general)
   END_RUNG
   RUNG wire#powerrail
      I_Contact( #statUnitStatus.mode.production )
      Contact( "Unit1.Em4.HmiInterface".cutter.sequence.monitoring.inStepIdle )
   END_RUNG wire#w1
   // the same network as SCL:
   #instFeedingRollAxisControlInterlockSummary(enableManualCmds := NOT #statUnitStatus.mode.production AND "Unit1.Em4.HmiInterface".cutter.sequence.monitoring.inStepIdle,   // "LER_AxisControl_InterlockSummary"
                           interlockSource := "Unit1.Em4.ControlNodes".cm.Interlock.feedingRoll.source,
                           moduleInterface := "Unit1.Em4.HmiInterface".cmFeedingRollAxisB,
                           controlNode := "Unit1.Em4.ControlNodes".cmFeedingRollAxisB,
                           interlockcGeneral => "Unit1.Em4.ControlNodes".cm.Interlock.feedingRoll.permit.general);
END_REGION

REGION Network 65: Call CM Feeding Roll B Axis (LBC_AxisControl)
   RUNG wire#powerrail
      #instCmFeedingRollAxisB(enable := wire#w1, parentReferenceDesignator := "Unit1.Em4.Config".em.referenceDesignator.combined, overrideVelocity :=, overrideVelocityPct :=, interlockGeneral := "Unit1.Em4.ControlNodes".cm.Interlock.feedingRoll.permit.general, interlockJogForward := "Unit1.Em4.ControlNodes".cm.Interlock.feedingRoll.permit.jogForward, interlockJogBackward := "Unit1.Em4.ControlNodes".cm.Interlock.feedingRoll.permit.jogBackward, enableManualCmds := #statEnableManualCmds, moduleAccessPoint := "Unit1.Em4.Config".moduleAccessPoint[2], axisNo :=, axis := "Unit1.Em4.Config".axis[2], master :=, cam :=, configuration := "Unit1.Em4.Config".cmFeedingRollAxisB, moduleInterface := "Unit1.Em4.HmiInterface".cmFeedingRollAxisB, controlNode := "Unit1.Em4.ControlNodes".cmFeedingRollAxisB, busy =>, actualPosition =>, actualSpeed =>)
   END_RUNG
   RUNG wire#powerrail
      Contact( #TRUE )
   END_RUNG wire#w1
   // the same network as SCL:
   #instCmFeedingRollAxisB(enable := #TRUE,   // "LBC_AxisControl_TecPlcCn"
                           parentReferenceDesignator := "Unit1.Em4.Config".em.referenceDesignator.combined,
                           interlockGeneral := "Unit1.Em4.ControlNodes".cm.Interlock.feedingRoll.permit.general,
                           interlockJogForward := "Unit1.Em4.ControlNodes".cm.Interlock.feedingRoll.permit.jogForward,
                           interlockJogBackward := "Unit1.Em4.ControlNodes".cm.Interlock.feedingRoll.permit.jogBackward,
                           enableManualCmds := #statEnableManualCmds,
                           moduleAccessPoint := "Unit1.Em4.Config".moduleAccessPoint[2],
                           axis := "Unit1.Em4.Config".axis[2],
                           configuration := "Unit1.Em4.Config".cmFeedingRollAxisB,
                           moduleInterface := "Unit1.Em4.HmiInterface".cmFeedingRollAxisB,
                           controlNode := "Unit1.Em4.ControlNodes".cmFeedingRollAxisB);
END_REGION

REGION Network 66: Call CM Feeding Roll B Axis (LER_ServoTorqueCal)
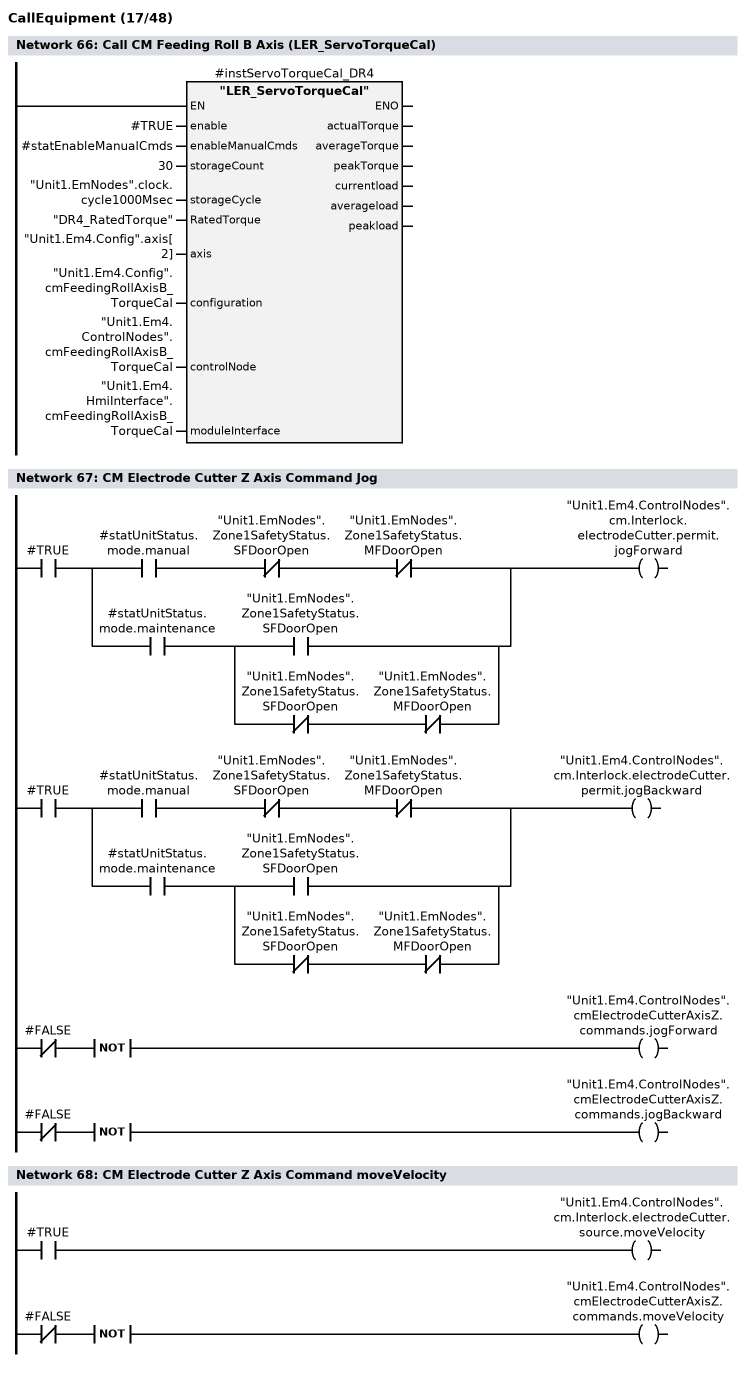
   RUNG wire#powerrail
      #instServoTorqueCal_DR4(enable := #TRUE, enableManualCmds := #statEnableManualCmds, storageCount := 30, storageCycle := "Unit1.EmNodes".clock.cycle1000Msec, RatedTorque := "DR4_RatedTorque", axis := "Unit1.Em4.Config".axis[2], configuration := "Unit1.Em4.Config".cmFeedingRollAxisB_TorqueCal, controlNode := "Unit1.Em4.ControlNodes".cmFeedingRollAxisB_TorqueCal, moduleInterface := "Unit1.Em4.HmiInterface".cmFeedingRollAxisB_TorqueCal, actualTorque =>, averageTorque =>, peakTorque =>, currentload =>, averageload =>, peakload =>)
   END_RUNG
   // the same network as SCL:
   #instServoTorqueCal_DR4(enable := #TRUE,   // "LER_ServoTorqueCal"
                           enableManualCmds := #statEnableManualCmds,
                           storageCount := 30,
                           storageCycle := "Unit1.EmNodes".clock.cycle1000Msec,
                           RatedTorque := "DR4_RatedTorque",
                           axis := "Unit1.Em4.Config".axis[2],
                           configuration := "Unit1.Em4.Config".cmFeedingRollAxisB_TorqueCal,
                           controlNode := "Unit1.Em4.ControlNodes".cmFeedingRollAxisB_TorqueCal,
                           moduleInterface := "Unit1.Em4.HmiInterface".cmFeedingRollAxisB_TorqueCal);
END_REGION

REGION Network 67: CM Electrode Cutter Z Axis Command Jog
   RUNG wire#powerrail
      Contact( #TRUE )
      wire#w1
      Contact( #statUnitStatus.mode.manual )
      I_Contact( "Unit1.EmNodes".Zone1SafetyStatus.SFDoorOpen )
      I_Contact( "Unit1.EmNodes".Zone1SafetyStatus.MFDoorOpen )
      wire#w2
      Coil( "Unit1.Em4.ControlNodes".cm.Interlock.electrodeCutter.permit.jogForward )
   END_RUNG
   RUNG wire#w1
      Contact( #statUnitStatus.mode.maintenance )
      wire#w3
      Contact( "Unit1.EmNodes".Zone1SafetyStatus.SFDoorOpen )
   END_RUNG wire#w2
   RUNG wire#w3
      I_Contact( "Unit1.EmNodes".Zone1SafetyStatus.SFDoorOpen )
      I_Contact( "Unit1.EmNodes".Zone1SafetyStatus.MFDoorOpen )
   END_RUNG wire#w2
   RUNG wire#powerrail
      Contact( #TRUE )
      wire#w4
      Contact( #statUnitStatus.mode.manual )
      I_Contact( "Unit1.EmNodes".Zone1SafetyStatus.SFDoorOpen )
      I_Contact( "Unit1.EmNodes".Zone1SafetyStatus.MFDoorOpen )
      wire#w5
      Coil( "Unit1.Em4.ControlNodes".cm.Interlock.electrodeCutter.permit.jogBackward )
   END_RUNG
   RUNG wire#w4
      Contact( #statUnitStatus.mode.maintenance )
      wire#w6
      Contact( "Unit1.EmNodes".Zone1SafetyStatus.SFDoorOpen )
   END_RUNG wire#w5
   RUNG wire#w6
      I_Contact( "Unit1.EmNodes".Zone1SafetyStatus.SFDoorOpen )
      I_Contact( "Unit1.EmNodes".Zone1SafetyStatus.MFDoorOpen )
   END_RUNG wire#w5
   RUNG wire#powerrail
      I_Contact( #FALSE )
      Not()
      Coil( "Unit1.Em4.ControlNodes".cmElectrodeCutterAxisZ.commands.jogForward )
   END_RUNG
   RUNG wire#powerrail
      I_Contact( #FALSE )
      Not()
      Coil( "Unit1.Em4.ControlNodes".cmElectrodeCutterAxisZ.commands.jogBackward )
   END_RUNG
   // the same network as SCL:
   "Unit1.Em4.ControlNodes".cm.Interlock.electrodeCutter.permit.jogForward := #TRUE AND ((#statUnitStatus.mode.manual AND NOT "Unit1.EmNodes".Zone1SafetyStatus.SFDoorOpen AND NOT "Unit1.EmNodes".Zone1SafetyStatus.MFDoorOpen) OR (#statUnitStatus.mode.maintenance AND ("Unit1.EmNodes".Zone1SafetyStatus.SFDoorOpen OR (NOT "Unit1.EmNodes".Zone1SafetyStatus.SFDoorOpen AND NOT "Unit1.EmNodes".Zone1SafetyStatus.MFDoorOpen))));
   "Unit1.Em4.ControlNodes".cm.Interlock.electrodeCutter.permit.jogBackward := #TRUE AND ((#statUnitStatus.mode.manual AND NOT "Unit1.EmNodes".Zone1SafetyStatus.SFDoorOpen AND NOT "Unit1.EmNodes".Zone1SafetyStatus.MFDoorOpen) OR (#statUnitStatus.mode.maintenance AND ("Unit1.EmNodes".Zone1SafetyStatus.SFDoorOpen OR (NOT "Unit1.EmNodes".Zone1SafetyStatus.SFDoorOpen AND NOT "Unit1.EmNodes".Zone1SafetyStatus.MFDoorOpen))));
   "Unit1.Em4.ControlNodes".cmElectrodeCutterAxisZ.commands.jogForward := NOT (NOT #FALSE);
   "Unit1.Em4.ControlNodes".cmElectrodeCutterAxisZ.commands.jogBackward := NOT (NOT #FALSE);
END_REGION

REGION Network 68: CM Electrode Cutter Z Axis Command moveVelocity
   RUNG wire#powerrail
      Contact( #TRUE )
      Coil( "Unit1.Em4.ControlNodes".cm.Interlock.electrodeCutter.source.moveVelocity )
   END_RUNG
   RUNG wire#powerrail
      I_Contact( #FALSE )
      Not()
      Coil( "Unit1.Em4.ControlNodes".cmElectrodeCutterAxisZ.commands.moveVelocity )
   END_RUNG
   // the same network as SCL:
   "Unit1.Em4.ControlNodes".cm.Interlock.electrodeCutter.source.moveVelocity := #TRUE;
   "Unit1.Em4.ControlNodes".cmElectrodeCutterAxisZ.commands.moveVelocity := NOT (NOT #FALSE);
END_REGION

REGION Network 69: CM Electrode Cutter Z Axis Command stop
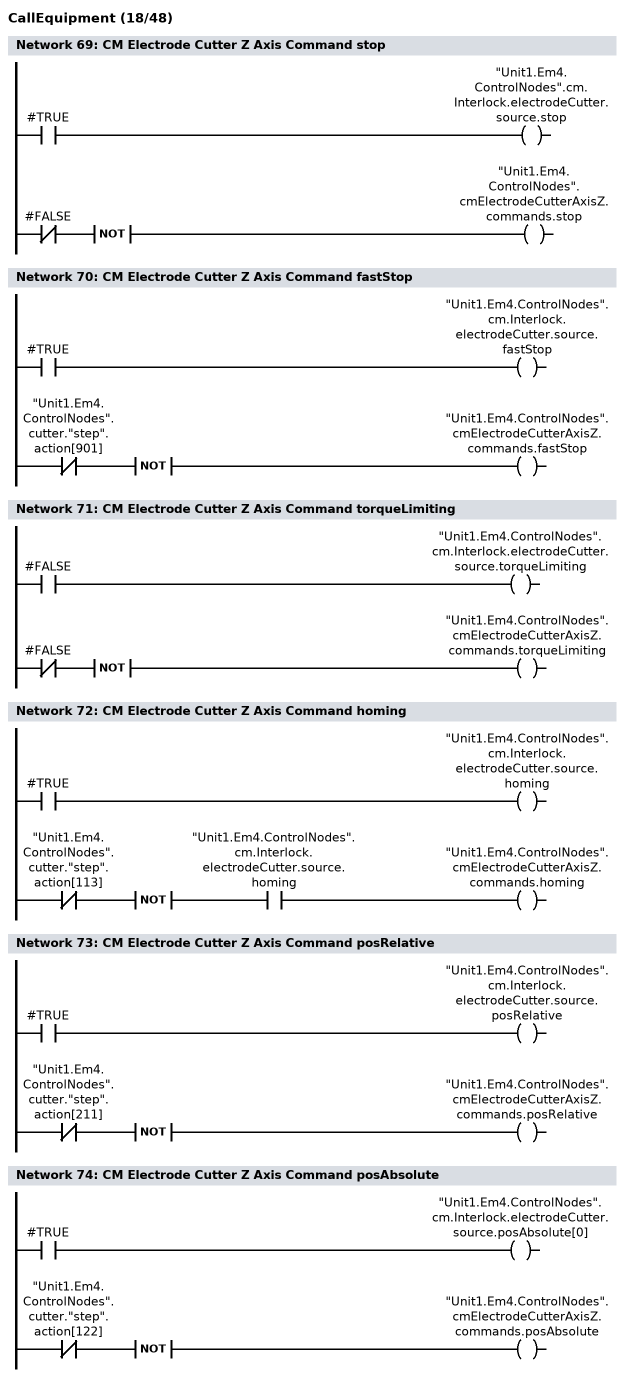
   RUNG wire#powerrail
      Contact( #TRUE )
      Coil( "Unit1.Em4.ControlNodes".cm.Interlock.electrodeCutter.source.stop )
   END_RUNG
   RUNG wire#powerrail
      I_Contact( #FALSE )
      Not()
      Coil( "Unit1.Em4.ControlNodes".cmElectrodeCutterAxisZ.commands.stop )
   END_RUNG
   // the same network as SCL:
   "Unit1.Em4.ControlNodes".cm.Interlock.electrodeCutter.source.stop := #TRUE;
   "Unit1.Em4.ControlNodes".cmElectrodeCutterAxisZ.commands.stop := NOT (NOT #FALSE);
END_REGION

REGION Network 70: CM Electrode Cutter Z Axis Command fastStop
   RUNG wire#powerrail
      Contact( #TRUE )
      Coil( "Unit1.Em4.ControlNodes".cm.Interlock.electrodeCutter.source.fastStop )
   END_RUNG
   RUNG wire#powerrail
      I_Contact( "Unit1.Em4.ControlNodes".cutter."step".action[901] )
      Not()
      Coil( "Unit1.Em4.ControlNodes".cmElectrodeCutterAxisZ.commands.fastStop )
   END_RUNG
   // the same network as SCL:
   "Unit1.Em4.ControlNodes".cm.Interlock.electrodeCutter.source.fastStop := #TRUE;
   "Unit1.Em4.ControlNodes".cmElectrodeCutterAxisZ.commands.fastStop := NOT (NOT "Unit1.Em4.ControlNodes".cutter."step".action[901]);
END_REGION

REGION Network 71: CM Electrode Cutter Z Axis Command torqueLimiting
   RUNG wire#powerrail
      Contact( #FALSE )
      Coil( "Unit1.Em4.ControlNodes".cm.Interlock.electrodeCutter.source.torqueLimiting )
   END_RUNG
   RUNG wire#powerrail
      I_Contact( #FALSE )
      Not()
      Coil( "Unit1.Em4.ControlNodes".cmElectrodeCutterAxisZ.commands.torqueLimiting )
   END_RUNG
   // the same network as SCL:
   "Unit1.Em4.ControlNodes".cm.Interlock.electrodeCutter.source.torqueLimiting := #FALSE;
   "Unit1.Em4.ControlNodes".cmElectrodeCutterAxisZ.commands.torqueLimiting := NOT (NOT #FALSE);
END_REGION

